// K2/std12k5/algoritms/YstavkiConfig
TYPE YstavkiConfig:
		{attribute 'symbol' := 'read'} 
	STRUCT
		blockkr1: (*REFERENCE TO*)  DiscretParametr (table:=ADR(YstTable)) ;//{name:блокировать самосдвиг крана 1}
		blockkr2:(*REFERENCE TO*) DiscretParametr (table:=ADR(YstTable));//{name:блокировать самосдвиг крана 2}
		blockkr3:(*REFERENCE TO*) DiscretParametr (table:=ADR(YstTable));//{name:блокировать самосдвиг крана 3}
		blockkr3b:(*REFERENCE TO*) DiscretParametr (table:=ADR(YstTable));//{name:блокировать самосдвиг крана 3б}
		blockkr4:(*REFERENCE TO*) DiscretParametr (table:=ADR(YstTable));//{name:блокировать самосдвиг крана 4}
		blockkr5:(*REFERENCE TO *)DiscretParametr (table:=ADR(YstTable));//{name:блокировать самосдвиг крана 5}
		blockkr6:(*REFERENCE TO *)DiscretParametr (table:=ADR(YstTable));//{name:блокировать самосдвиг крана 6}
		Block_kr4_alg:DiscretParametr (table:=ADR(YstTable));
		Block_kr1_alg:DiscretParametr (table:=ADR(YstTable));
		Block_kr2_alg:DiscretParametr (table:=ADR(YstTable));
		Block_kr3_alg:DiscretParametr (table:=ADR(YstTable));
		Block_kr3b_alg:DiscretParametr (table:=ADR(YstTable));
		Block_kr5_alg:DiscretParametr (table:=ADR(YstTable));
		Block_kr6_alg:DiscretParametr (table:=ADR(YstTable));
		
		block_OPC_cmd:DiscretParametr (table:=ADR(YstTable));
		
		////////////////////ПС по СИП//////////////////////////////////////////////////////
		SIp_T1: SIP_PS (table:=ADR(YstTable)):=(ai:= ai.TOpornogoPodshipnikaEDT_1);
		
		SIp_T2: SIP_PS (table:=ADR(YstTable)):=(ai:= ai.TOpornoYpornogoPodshipnikaEDT_2);
		
		SIp_T3: SIP_PS (table:=ADR(YstTable)):=(ai:= ai.TOpornoYpornogoPodshipnikaKolesaRedEDT_3);
		
		SIp_T4: SIP_PS (table:=ADR(YstTable)):=(ai:= ai.TOpornoYpornogoPodshipnikaKolesaRedHT_4);
		
		SIp_T5: SIP_PS (table:=ADR(YstTable)):=(ai:= ai.TOpornogoPodshipnikaShesterniReduktoraT_5);
		
		SIp_T6: SIP_PS (table:=ADR(YstTable)):=(ai:= ai.TOpornogoPodshipnikaReduktoraHT_6);
		
		SIp_T7_1: SIP_PS (table:=ADR(YstTable)):=(ai:= ai.TOpornoYpornogoPodshipnikaNagnetateljaT_7_1);
		
		SIp_T7_2: SIP_PS (table:=ADR(YstTable)):=(ai:= ai.TOpornoYpornogoPodshipnikaNagnetateljaT_7_2);
		
		SIp_T8_1: SIP_PS (table:=ADR(YstTable)):=(ai:= ai.TOpornoYpornogoPodshipnikaSvobodnogoKoncaNT_8_1);
		
		SIp_T8_2: SIP_PS (table:=ADR(YstTable)):=(ai:= ai.TOpornoYpornogoPodshipnikaSvobodnogoKoncaNT_8_2);
		
		SIp_T9_1: SIP_PS (table:=ADR(YstTable)):=(ai:= ai.TYpornogoPodshipnikaRavKolodokHT_9_1	);
		
		SIp_T9_2: SIP_PS (table:=ADR(YstTable)):=(ai:= ai.TYpornogoPodshipnikaRavKolodokHT_9_2	);
		
		SIp_T10_1: SIP_PS (table:=ADR(YstTable)):=(ai:= ai.TYpornogoPodshipnikaNerabKolodokHT_10_1	);
		
		SIp_T10_2: SIP_PS (table:=ADR(YstTable)):=(ai:= ai.TYpornogoPodshipnikaNerabKolodokHT_10_2	);
		
		SIp_T_Vyhode_N: SIP_PS (table:=ADR(YstTable)):=(ai:= ai.TgazaNaVyhodeH);
		
		SIp_T_Posle_AVOM: SIP_PS (table:=ADR(YstTable)):=(ai:= ai.TMaslaPosleAVOM);
		
		SIp_T_Masla_MB: SIP_PS (table:=ADR(YstTable)):=(ai:= ai.TMaslaMB);
		
		SIp_T_Masla_TEN: SIP_PS (table:=ADR(YstTable)):=(ai:= ai.TMaslaMB_TEN);
		
		////////////////////НАРАБОТКА//////////////////////////////////////////////////////
		
		nu1_narab: nu1 (table:=ADR(YstTable));		
		nu2_narab: nu2 (table:=ADR(YstTable));
		//pns_narab: pns_ (table:=ADR(YstTable));
		Work_HRS: work (table:=ADR(YstTable));
		Pusk_times: pusk (table:=ADR(YstTable));
		AO_times: AO (table:=ADR(YstTable));
		NO_times: NO (table:=ADR(YstTable));
		EO_times: EO (table:=ADR(YstTable));
		//CMN_Narab:CMN (table:=ADR(YstTable));
		//Kalorifer_AVOM_Narab: Kalorifer_AVOM (table:=ADR(YstTable));
		//TEN_Kollectora_narab: TEN_Kollectora (table:=ADR(YstTable));
	//	TEN_MB_Narab:			TEN_MB (table:=ADR(YstTable));
		////////////////////Уставки//////////////////////////////////////////////////////
		YstPNS_YP:  AutoPNS_YP (table:=ADR(YstTable));
		YstPNS_YT:  AutoPNS_YT (table:=ADR(YstTable));
		
		Yst_Vkl_TEN:	AutoTEN_YP (table:=ADR(YstTable));
		Yst_Vykl_TEN:	AutoTEN_YT (table:=ADR(YstTable));
		
		Yst_AVOM_T1:	T1_AVOM (table:=ADR(YstTable));
		Yst_AVOM_T2:	T2_AVOM (table:=ADR(YstTable));
		Yst_AVOM_T3:	T3_AVOM (table:=ADR(YstTable));
		Yst_AVOM_T4:	T4_AVOM (table:=ADR(YstTable));
		
		Yst_Tvkl_AVOM1:	Tvkl_AVOM1 (table:=ADR(YstTable));
		Yst_Tvkl_AVOM2:	Tvkl_AVOM2 (table:=ADR(YstTable));
		Yst_Tvkl_AVOM3:	Tvkl_AVOM3 (table:=ADR(YstTable));
		Yst_Tvkl_AVOM4:	Tvkl_AVOM4 (table:=ADR(YstTable));
		
		Yst_Tvykl_AVOM1:	Tvykl_AVOM1 (table:=ADR(YstTable));
		Yst_Tvykl_AVOM2:	Tvykl_AVOM2 (table:=ADR(YstTable));
		Yst_Tvykl_AVOM3:	Tvykl_AVOM3 (table:=ADR(YstTable));
		Yst_Tvykl_AVOM4:	Tvykl_AVOM4 (table:=ADR(YstTable));
		
		Yst_DTvykl_AVOM1:	Delta_Vykl_AVOM1 (table:=ADR(YstTable));
		Yst_DTvykl_AVOM2:	Delta_Vykl_AVOM2 (table:=ADR(YstTable));
		Yst_DTvykl_AVOM3:	Delta_Vykl_AVOM3 (table:=ADR(YstTable));
		Yst_DTvykl_AVOM4:	Delta_Vykl_AVOM4 (table:=ADR(YstTable));
		
		num_Avom:			Number_Of_Avom (table:=ADR(YstTable));
		
		////////////////////Управляющие сигналы//////////////////////////////////////////////////////
		//{name:рассогласование аналогов и дискрета по dPм-г}
		dPmg_Rassogl: Rassoglasovanie_dPmg (table:=ADR(YstTable)):=(di:=im.PerepadDavlenieMasloGaz_Less100, ai:=AI.PerepadDavlenieMasloGaz);
		dP_Konf_kr1:DiscretParametr (table:=ADR(YstTable));	
		dP_Konf_kr2:DiscretParametr (table:=ADR(YstTable));	
		(*sip_t1_new:SEt_New_SIP (table:=ADR(YstTable)):=(Ai:=ai.TOpornogoPodshipnikaEDT_1, n:= 0);*)
	END_STRUCT
END_TYPE

// lowLevel_ecl/kontroller/extSources/AnalogsProcessing
TYPE AnalogsProcessing :
(
	AVERAGEVALUE,
	MAXVALUE,
	MINVALUE,
	MEDIANVALUE
);
END_TYPE

// lowLevel_ecl/Common/table/TableDescriptor
TYPE TableDescriptor :
STRUCT
	head:POINTER TO BaseObject:=0;
	tail:POINTER TO BaseObject:=0;
END_STRUCT
END_TYPE

// lowLevel_ecl/im/sectionSwitch/basketStats
TYPE basketStats :
(
	BASKET_NOTDEFINED:=0,
	BASKET_ROLLEDIN:=1,
	BASKET_ROLLEDOUT:=2,
	BASKET_TRANSITIONAL:=3,
	BASKET_ERROR:=4,
	BASKET_TEST:=5
) BYTE;
END_TYPE

// lowLevel_ecl/kontroller/modbus/MbAiWordOrder
TYPE MbAiWordOrder :
(
	AiWordOrder12 := 0,
	AiWordOrder21 := 1
);
END_TYPE

// lowLevel_ecl/kontroller/modbus/MbKontrollerRole
TYPE MbKontrollerRole :
(
	MK_DONTKNOWN,
	MK_MASTER,
	MK_SLAVE
);
END_TYPE

// lowLevel_ecl/kontroller/modbus/Sources/FloatAsWords
TYPE FloatAsWords :
UNION
	fValue:REAL;
	wValue:ARRAY[0..1]OF WORD;
	dwValue:DWORD;
	bValue:ARRAY[0..4]OF BYTE;
END_UNION
END_TYPE

// lowLevel_ecl/kontroller/modbus/UsedByteMBSource
TYPE UsedByteMBSource :
(
	LB,
	HB
);
END_TYPE

// K1/std12k5/hardwareConfig/defines/hwC
	{attribute 'symbol' := 'readwrite'}
VAR_GLOBAL
	//SIP:	SIp_Yst (table:=0);
		{attribute 'symbol' := 'none'}
	kontrollers:TableDescriptor;
		{attribute 'symbol' := 'read'}
///	kontroller:elpk04(table:=ADR(kontrollers)):=(mlpConfig:='C:\\ELPK04\\Mlp2 2015-04-07\\MLP Projects\\1.mlp');
	kontroller:elpk04(table:=ADR(kontrollers)):=(mlpConfig:='\Storage Card\3s\RWHxxx.INI');// не должно находить такой файл никогда !!!
	di:DiConfig;
	ai:AiConfig;
	od:DOConfig;
	{attribute 'symbol' := 'none'}
	ao:AOConfig;
	//{attribute 'symbol' := 'none'}
	//mb:MbsConfig;

END_VAR

// K1/std12k5/logicConfig/defines/logicConfig
	{attribute 'symbol' := 'readwrite'}
VAR_GLOBAL
	{attribute 'symbol' := 'none'}
	imTable:TableDescriptor;
	
	{attribute 'symbol' := 'none'}
	iAmTrue:everifingTrue(table:=0);//Затычка из DiSource. Всегда возвращает одни и теже комбинации значения и достоверности
	OPC_Imit: Imit_OPC (table:=0);
	Im:ImConfig;
	{attribute 'symbol' := 'none'}
	Off_Q:All_Quation_Off (table:=0);
		{attribute 'symbol' := 'none'}
	PPU_Init_:PPU_Init (table:=0);
END_VAR

// K1/std12k5/algoritms/defines/algoritmsConf
	{attribute 'symbol' := 'readwrite'}
VAR_GLOBAL
	{attribute 'symbol' := 'none'}
	YstTable:TableDescriptor;
	Ystavki: YstavkiConfig;
	algManager:AlgoritmsManager(table:=0);
	algoritms:algoritmsConfig;
	{attribute 'symbol' := 'none'}
	protectManager:ProtectionManager (table:=0);
	protections:ProtectionsConfig;
	
	
END_VAR

// lowLevel_ecl/kontroller/mlp/FAUs
{attribute 'symbol' := 'none'}
VAR_GLOBAL
	
DIn_ 	:	ARRAY [0..255] 	OF DIn_s;		//	Сигнализация и неисправности дискретных входов (номер в массиве соответствует адресу конфигурации в MLP)
											//	f	:	WORD	;	//	bit-0 присутствие в проекте MLP. 1-есть, 0 -нет
																	//	bit-1 тип модуля 1-выходной, 0 -входной
																	//	bit-2 достоверность 1- достоверно,0- не достоверно 
											//	val	:	WORD	;	//	Контроль канала
																	//	Каждая цепь 2 бита
	                												//	00 - обыв цепи
																	//	01 - недостоверно
																	//	10 - контакт разомкнут
																	//	11 - контакт замкнут	

											//	DIn[63].val - меняющееся число для проверки связи с основным МЛП (задается в MLP)
											//	если	DIn[64].val = 7 - есть связь с BS-1 (задается в MLP)
											//	если	DIn[65].val = 7 - есть связь с BS-2 (задается в MLP)
											//	если	DIn[66].val = 7 - есть связь с BS-3 (задается в MLP)
											//	если	DIn[67].val = 7 - есть связь с BS-4 (задается в MLP)
																					
																	
AIn_ 	:	ARRAY [0..255] 	OF AIn_s;		//	Значение и неисправности аналоговых входов (номер в массиве соответствует адресу конфигурации в MLP)
											//	f	:	DWORD	;	//	bit-0 присутствие в проекте MLP. 1-есть, 0 –нет
																	//	bit-1 тип модуля 1-выходной, 0 -входной
																	//	bit-2 достоверность 1- достоверно,0- не достоверно. Диагностика общая: и по диапазонам измерения, и собственная по каналу модуля.
																	//	bit-3 размерность сигнала 1- в физических величинах,0- значение тока (0-20100)
																	//	bit-4 1- ниже нижней границы,0 - выше нижней границы
																	//	bit-5 1- выше верхней границы,0 - ниже верхней границы
																	//	bit-6 1- общий бит отказа канала( по ИЛИ Not(bit2), bit4, bit5)
											//	val	:	REAL	;	//	Значение аналогового входа 4-20мА - 40000-20000 

Dout_	:	ARRAY [0..255] 	OF WORD;		//	Массив дискретных выходов (один бит - один выход, одно слово - один модуль) (номер в массиве соответствует адресу конфигурации в MLP)
Din_Dout: 	ARRAY [0..255] 	OF sDIN_DOUT;	//	Массив неисправностей дискретных выходов
											//	s_Aux	:	WORD	;	//	bit-0 присутствие 1-есть, 0 -нет (привязка в конфигурации MLP)
																		//	bit-1 тип модуля 1-выходной, 0 -входной
																		//	bit-2 достоверность 1- достоверно,0- не достоверно
									  		//	kcc		:	WORD	;   //	Контроль Целостности Цепи - КЦЦ
																		//	каждая цепь 2 бита
																		//	00 - неизвестно или обрыв цепи
																		//	01 - есть Целостность Цепи
																		//	10 - есть ток
																		//	11 - КЗ
											//	kk		:	WORD	;	//	Контроль выхода команды - КК
																		//	каждая цепь 2 бита
																		//	00 - не бывает
																		//	01 - пассивное состояние
																		//	10 - активное (есть выход)состояние
																		//	11 - ошибка выхода команды 
									  		//	value_cc:	WORD	;	//	содержимое выходных регистров 

Aout_ 	:	ARRAY [0..255] 	OF REAL;		//	Массив аналоговых выходов (номер в массиве соответствует адресу конфигурации в MLP)
Ain_Aout:	ARRAY [0..255] 	OF sAIN_AOUT;	//	Массив неисправностей аналоговых выходов
											//	s_Aux	:	WORD	;	//	bit-0 присутствие 1-есть, 0 -нет
																		//	bit-1 тип модуля 1-выходной, 0 -входной
																		//	bit-2 достоверность 1- достоверно,0- не достоверно
																		//	s_value	:	REAL	;	//	Действительный (измеренный) выходной ток 4-20мА - 4000-20000

Diag_ 	:	ARRAY [0..63]	OF WORD;		//	массив неисправностей модулей
																		//	2 бита на 1 модуль
																		//	00 - ok
																		//	01 - нет модуля
																		//	10 - нулевые данные
																		//	11 - нет связи с модулем
END_VAR

// K1/std12k5/Elpk_03_02/GVL_COMMON
VAR_GLOBAL

//////////////////// П Е Р Е М Е Н Н Ы Е //////////////////////////////////////////////////////////////////////////////

	DI_K:ARRAY[0..255] OF T_DI03{WORD};
	AI_K:ARRAY[0..255] OF T_AI03{WORD};
	DO_K:ARRAY[0..255] OF T_DO03;
	
	MODULES03:ARRAY[1..16] OF T_DIAGNOSTIC03;
	IMIT_F:	WORD:= 0;	//16#55AA;







//	Глобальные переменные для резервирования
	H1:RTS_IEC_HANDLE;// pointer to byte
	S1:Com_Settings;
	S1ex:Com_SettingsEX;

	
//	Глобальные переменные для OPC
   {attribute 'displaymode':='hex'}
	BMPERR_I:WORD;		// внутреннее использование
   {attribute 'displaymode':='hex'}
	MxStatus_I:WORD;		// внутреннее использование
   {attribute 'displaymode':='hex'}
	MxMode_O:WORD;		// внутреннее использование
   {attribute 'displaymode':='hex'}
	BMPPRES_I:WORD;		// внутреннее использование






	



(*
//////////////////////////////////////////////////////////////////////
//This gobal variable list is received via the network.
//Sender: GVL2N_REZ [UP2: PLC Logic: Application]
//Protocol: UDP
//	Глобальные переменные для резервирования - это должно быть в глоб списке передачи К2
	PilaK2_O:WORD;
	StatusK2_O:WORD;
	ReadyK2_O:WORD;
////////////////////////////////////////////////////////////////////////
*)





//////////////////////////////////////////////////////////////////////
//This gobal variable list is received via the network.
//Sender: GVL1IMIT_to [Imitator1: PLC Logic: Application]
//Protocol: UDP
//	Глобальные переменные для моего имитатора. Должно быть в NVL1_from_IMIT
//
//
//   {attribute 'displaymode':='hex'}
//	Imitator_Code:WORD:=16#55AA;// код наличия имитатора - пересылается из имитатора в контроллеры!!!
   {attribute 'displaymode':='hex'}
	Imitator_Code:WORD:=16#0;// код наличия имитатора - пересылается из имитатора в контроллеры!!!

	// аналоговые входы нумеруем от 1
	AIs_Im:ARRAY[0..100] OF WORD;// рассылка из имитатора
	// дискретные входы нумеруем от 1
   {attribute 'displaymode':='hex'}
	DIs_Im:ARRAY[0..30] OF WORD;// рассылка из имитатора
(*
	// пока не используется в имитаторе !!!	
	// диагностика контроллера №1 
   {attribute 'displaymode':='hex'}
	NodeErr1_UP1_Im:WORD;// рассылка из имитатора
   {attribute 'displaymode':='hex'}
	NodeErr2_UP1_Im:WORD;// рассылка из имитатора
   {attribute 'displaymode':='hex'}
	NodeErr3_UP1_Im:WORD;// рассылка из имитатора
   {attribute 'displaymode':='hex'}
	NodeErr4_UP1_Im:WORD;// рассылка из имитатора
   {attribute 'displaymode':='hex'}
	NodeErr5_UP1_Im:WORD;// рассылка из имитатора
   {attribute 'displaymode':='hex'}
	NodeErr6_UP1_Im:WORD;// рассылка из имитатора
   {attribute 'displaymode':='hex'}
	NodeErr7_UP1_Im:WORD;// рассылка из имитатора
   {attribute 'displaymode':='hex'}
	NodeErr8_UP1_Im:WORD;// рассылка из имитатора
   {attribute 'displaymode':='hex'}
	NodeErr9_UP1_Im:WORD;// рассылка из имитатора
   {attribute 'displaymode':='hex'}
	NodeErr10_UP1_Im:WORD;// рассылка из имитатора
   {attribute 'displaymode':='hex'}
	NodeErr11_UP1_Im:WORD;// рассылка из имитатора
   {attribute 'displaymode':='hex'}
	NodeErr12_UP1_Im:WORD;// рассылка из имитатора
   {attribute 'displaymode':='hex'}
	NodeErr13_UP1_Im:WORD;// рассылка из имитатора
   {attribute 'displaymode':='hex'}
	NodeErr14_UP1_Im:WORD;// рассылка из имитатора
   {attribute 'displaymode':='hex'}
	NodeErr15_UP1_Im:WORD;// рассылка из имитатора
   {attribute 'displaymode':='hex'}
	NodeErr16_UP1_Im:WORD;// рассылка из имитатора
   {attribute 'displaymode':='hex'}
	BMPERR_UP1_Im:WORD;// рассылка из имитатора
   {attribute 'displaymode':='hex'}
	BMPPRES_UP1_Im:WORD;// рассылка из имитатора

	// диагностика контроллера №2 
   {attribute 'displaymode':='hex'}
	NodeErr1_UP2_Im:WORD;// рассылка из имитатора
   {attribute 'displaymode':='hex'}
	NodeErr2_UP2_Im:WORD;// рассылка из имитатора
   {attribute 'displaymode':='hex'}
	NodeErr3_UP2_Im:WORD;// рассылка из имитатора
   {attribute 'displaymode':='hex'}
	NodeErr4_UP2_Im:WORD;// рассылка из имитатора
   {attribute 'displaymode':='hex'}
	NodeErr5_UP2_Im:WORD;// рассылка из имитатора
   {attribute 'displaymode':='hex'}
	NodeErr6_UP2_Im:WORD;// рассылка из имитатора
   {attribute 'displaymode':='hex'}
	NodeErr7_UP2_Im:WORD;// рассылка из имитатора
   {attribute 'displaymode':='hex'}
	NodeErr8_UP2_Im:WORD;// рассылка из имитатора
   {attribute 'displaymode':='hex'}
	NodeErr9_UP2_Im:WORD;// рассылка из имитатора
   {attribute 'displaymode':='hex'}
	NodeErr10_UP2_Im:WORD;// рассылка из имитатора
   {attribute 'displaymode':='hex'}
	NodeErr11_UP2_Im:WORD;// рассылка из имитатора
   {attribute 'displaymode':='hex'}
	NodeErr12_UP2_Im:WORD;// рассылка из имитатора
   {attribute 'displaymode':='hex'}
	NodeErr13_UP2_Im:WORD;// рассылка из имитатора
   {attribute 'displaymode':='hex'}
	NodeErr14_UP2_Im:WORD;// рассылка из имитатора
   {attribute 'displaymode':='hex'}
	NodeErr15_UP2_Im:WORD;// рассылка из имитатора
   {attribute 'displaymode':='hex'}
	NodeErr16_UP2_Im:WORD;// рассылка из имитатора
   {attribute 'displaymode':='hex'}
	BMPERR_UP2_Im:WORD;// рассылка из имитатора
   {attribute 'displaymode':='hex'}
	BMPPRES_UP2_Im:WORD;// рассылка из имитатора
*)

END_VAR

// K1/std12k5/Elpk_03_02/GVL1N_REZ
VAR_GLOBAL
//	Глобальные переменные для резервирования
	PilaK1_O:WORD;
	StatusK1_O:WORD;
	ReadyK1_O:WORD;
		

END_VAR

// K1/std12k5/Elpk_03_02/GVLOPC
VAR_GLOBAL
//					
	LifeCnt:WORD;	// Пила жизни из контроллера: на каждом цикле +1 в диапазоне 0..1023
	
// диагностика контроллера	
   {attribute 'displaymode':='hex'}
	NodeErr1_K:WORD;	// OPC	
   {attribute 'displaymode':='hex'}
	NodeErr2_K:WORD;	// OPC
   {attribute 'displaymode':='hex'}
	NodeErr3_K:WORD;	// OPC
   {attribute 'displaymode':='hex'}
	NodeErr4_K:WORD;	// OPC
   {attribute 'displaymode':='hex'}
	NodeErr5_K:WORD;	// OPC
   {attribute 'displaymode':='hex'}
	NodeErr6_K:WORD;	// OPC
   {attribute 'displaymode':='hex'}
	NodeErr7_K:WORD;	// OPC
   {attribute 'displaymode':='hex'}
	NodeErr8_K:WORD;	// OPC
   {attribute 'displaymode':='hex'}
	NodeErr9_K:WORD;	// OPC
   {attribute 'displaymode':='hex'}
	NodeErr10_K:WORD;	// OPC
   {attribute 'displaymode':='hex'}
	NodeErr11_K:WORD;	// OPC
   {attribute 'displaymode':='hex'}
	NodeErr12_K:WORD;	// OPC
   {attribute 'displaymode':='hex'}
	NodeErr13_K:WORD;	// OPC
   {attribute 'displaymode':='hex'}
	NodeErr14_K:WORD;	// OPC
   {attribute 'displaymode':='hex'}
	NodeErr15_K:WORD;	// OPC
   {attribute 'displaymode':='hex'}
	NodeErr16_K:WORD;	// OPC

   {attribute 'displaymode':='hex'}
	CfgErr1_K:WORD;	// OPC	
   {attribute 'displaymode':='hex'}
	CfgErr2_K:WORD;	// OPC	
   {attribute 'displaymode':='hex'}
	CfgErr3_K:WORD;	// OPC	
   {attribute 'displaymode':='hex'}
	CfgErr4_K:WORD;	// OPC	
   {attribute 'displaymode':='hex'}
	CfgErr5_K:WORD;	// OPC	
   {attribute 'displaymode':='hex'}
	CfgErr6_K:WORD;	// OPC	
   {attribute 'displaymode':='hex'}
	CfgErr7_K:WORD;	// OPC	
   {attribute 'displaymode':='hex'}
	CfgErr8_K:WORD;	// OPC	
   {attribute 'displaymode':='hex'}
	CfgErr9_K:WORD;	// OPC	
   {attribute 'displaymode':='hex'}
	CfgErr10_K:WORD;	// OPC	
   {attribute 'displaymode':='hex'}
	CfgErr11_K:WORD;	// OPC	
   {attribute 'displaymode':='hex'}
	CfgErr12_K:WORD;	// OPC	
   {attribute 'displaymode':='hex'}
	CfgErr13_K:WORD;	// OPC	
   {attribute 'displaymode':='hex'}
	CfgErr14_K:WORD;	// OPC	
   {attribute 'displaymode':='hex'}
	CfgErr15_K:WORD;	// OPC	
   {attribute 'displaymode':='hex'}
	CfgErr16_K:WORD;	// OPC	




	
	
	
   {attribute 'displaymode':='hex'}
	BMPERR_K:WORD;	// OPC
   {attribute 'displaymode':='hex'}
	BMPPRES_K:WORD;	// OPC

   ///{attribute 'displaymode':='hex'}
	///DiagCnt_K:WORD;	// Пила диагностики из контроллера: на каждом цикле +1 в мл.байте и № контроллера в ст.байте
	
	
	
	// переменная master для ОРС-сервера
	MasterOPC_ST:BOOL;// ОРС-сервер читает переменную и если TRUE, то берет данные из этого контроллера
	LifeCntOPC:DWORD;// ОРС-сервер, если работает - записывает счетчик в переменную; если не работает- счетчик не изменяется




END_VAR

// K2/std12k5/hardwareConfig/defines/hwC
	{attribute 'symbol' := 'readwrite'}
VAR_GLOBAL
//	SIP:	SIp_Yst (table:=0);
		{attribute 'symbol' := 'none'}
	kontrollers:TableDescriptor;
		{attribute 'symbol' := 'read'}
///	kontroller:elpk04(table:=ADR(kontrollers)):=(mlpConfig:='C:\\ELPK04\\Mlp2 2015-04-07\\MLP Projects\\1.mlp');
	kontroller:elpk04(table:=ADR(kontrollers)):=(mlpConfig:='\Storage Card\3s\RWHxxx.INI');// не должно находить такой файл никогда !!!
	di:DiConfig;
	ai:AiConfig;
	od:DOConfig;
	{attribute 'symbol' := 'none'}
	ao:AOConfig;
//	{attribute 'symbol' := 'none'}
	//mb:MbsConfig;

END_VAR

// K2/std12k5/logicConfig/defines/logicConfig
	{attribute 'symbol' := 'readwrite'}
VAR_GLOBAL
	{attribute 'symbol' := 'none'}
	imTable:TableDescriptor;
	
	{attribute 'symbol' := 'none'}
	iAmTrue:everifingTrue(table:=0);//Затычка из DiSource. Всегда возвращает одни и теже комбинации значения и достоверности
	OPC_Imit: Imit_OPC (table:=0);
	Im:ImConfig;
	{attribute 'symbol' := 'none'}
	Off_Q:All_Quation_Off (table:=0);
		{attribute 'symbol' := 'none'}
	PPU_Init_:PPU_Init (table:=0);
END_VAR

// K2/std12k5/algoritms/defines/algoritmsConf
	{attribute 'symbol' := 'readwrite'}
VAR_GLOBAL
	{attribute 'symbol' := 'none'}
	YstTable:TableDescriptor;
	Ystavki: YstavkiConfig;
	algManager:AlgoritmsManager(table:=0);
	algoritms:algoritmsConfig;
	{attribute 'symbol' := 'none'}
	protectManager:ProtectionManager (table:=0);
	protections:ProtectionsConfig;
	
	
END_VAR

// K2/std12k5/Elpk_03_02/GVL_COMMON
VAR_GLOBAL

//////////////////// П Е Р Е М Е Н Н Ы Е //////////////////////////////////////////////////////////////////////////////

	DI_K:ARRAY[0..255] OF T_DI03{WORD};
	AI_K:ARRAY[0..255] OF T_AI03{WORD};
	DO_K:ARRAY[0..255] OF T_DO03;
	
	MODULES03:ARRAY[1..16] OF T_DIAGNOSTIC03;
	IMIT_F:	WORD:= 0;	//16#55AA;







//	Глобальные переменные для резервирования
	H1:RTS_IEC_HANDLE;// pointer to byte
	S1:Com_Settings;
	S1ex:Com_SettingsEX;

	
//	Глобальные переменные для OPC
   {attribute 'displaymode':='hex'}
	BMPERR_I:WORD;		// внутреннее использование
   {attribute 'displaymode':='hex'}
	MxStatus_I:WORD;		// внутреннее использование
   {attribute 'displaymode':='hex'}
	MxMode_O:WORD;		// внутреннее использование
   {attribute 'displaymode':='hex'}
	BMPPRES_I:WORD;		// внутреннее использование






	



(*
//////////////////////////////////////////////////////////////////////
//This gobal variable list is received via the network.
//Sender: GVL2N_REZ [UP2: PLC Logic: Application]
//Protocol: UDP
//	Глобальные переменные для резервирования - это должно быть в глоб списке передачи К2
	PilaK2_O:WORD;
	StatusK2_O:WORD;
	ReadyK2_O:WORD;
////////////////////////////////////////////////////////////////////////
*)





//////////////////////////////////////////////////////////////////////
//This gobal variable list is received via the network.
//Sender: GVL1IMIT_to [Imitator1: PLC Logic: Application]
//Protocol: UDP
//	Глобальные переменные для моего имитатора. Должно быть в NVL1_from_IMIT
//
//
//   {attribute 'displaymode':='hex'}
//	Imitator_Code:WORD:=16#55AA;// код наличия имитатора - пересылается из имитатора в контроллеры!!!
   {attribute 'displaymode':='hex'}
	Imitator_Code:WORD:=16#0;// код наличия имитатора - пересылается из имитатора в контроллеры!!!

	// аналоговые входы нумеруем от 1
	AIs_Im:ARRAY[0..100] OF WORD;// рассылка из имитатора
	// дискретные входы нумеруем от 1
   {attribute 'displaymode':='hex'}
	DIs_Im:ARRAY[0..30] OF WORD;// рассылка из имитатора
(*
	// пока не используется в имитаторе !!!	
	// диагностика контроллера №1 
   {attribute 'displaymode':='hex'}
	NodeErr1_UP1_Im:WORD;// рассылка из имитатора
   {attribute 'displaymode':='hex'}
	NodeErr2_UP1_Im:WORD;// рассылка из имитатора
   {attribute 'displaymode':='hex'}
	NodeErr3_UP1_Im:WORD;// рассылка из имитатора
   {attribute 'displaymode':='hex'}
	NodeErr4_UP1_Im:WORD;// рассылка из имитатора
   {attribute 'displaymode':='hex'}
	NodeErr5_UP1_Im:WORD;// рассылка из имитатора
   {attribute 'displaymode':='hex'}
	NodeErr6_UP1_Im:WORD;// рассылка из имитатора
   {attribute 'displaymode':='hex'}
	NodeErr7_UP1_Im:WORD;// рассылка из имитатора
   {attribute 'displaymode':='hex'}
	NodeErr8_UP1_Im:WORD;// рассылка из имитатора
   {attribute 'displaymode':='hex'}
	NodeErr9_UP1_Im:WORD;// рассылка из имитатора
   {attribute 'displaymode':='hex'}
	NodeErr10_UP1_Im:WORD;// рассылка из имитатора
   {attribute 'displaymode':='hex'}
	NodeErr11_UP1_Im:WORD;// рассылка из имитатора
   {attribute 'displaymode':='hex'}
	NodeErr12_UP1_Im:WORD;// рассылка из имитатора
   {attribute 'displaymode':='hex'}
	NodeErr13_UP1_Im:WORD;// рассылка из имитатора
   {attribute 'displaymode':='hex'}
	NodeErr14_UP1_Im:WORD;// рассылка из имитатора
   {attribute 'displaymode':='hex'}
	NodeErr15_UP1_Im:WORD;// рассылка из имитатора
   {attribute 'displaymode':='hex'}
	NodeErr16_UP1_Im:WORD;// рассылка из имитатора
   {attribute 'displaymode':='hex'}
	BMPERR_UP1_Im:WORD;// рассылка из имитатора
   {attribute 'displaymode':='hex'}
	BMPPRES_UP1_Im:WORD;// рассылка из имитатора

	// диагностика контроллера №2 
   {attribute 'displaymode':='hex'}
	NodeErr1_UP2_Im:WORD;// рассылка из имитатора
   {attribute 'displaymode':='hex'}
	NodeErr2_UP2_Im:WORD;// рассылка из имитатора
   {attribute 'displaymode':='hex'}
	NodeErr3_UP2_Im:WORD;// рассылка из имитатора
   {attribute 'displaymode':='hex'}
	NodeErr4_UP2_Im:WORD;// рассылка из имитатора
   {attribute 'displaymode':='hex'}
	NodeErr5_UP2_Im:WORD;// рассылка из имитатора
   {attribute 'displaymode':='hex'}
	NodeErr6_UP2_Im:WORD;// рассылка из имитатора
   {attribute 'displaymode':='hex'}
	NodeErr7_UP2_Im:WORD;// рассылка из имитатора
   {attribute 'displaymode':='hex'}
	NodeErr8_UP2_Im:WORD;// рассылка из имитатора
   {attribute 'displaymode':='hex'}
	NodeErr9_UP2_Im:WORD;// рассылка из имитатора
   {attribute 'displaymode':='hex'}
	NodeErr10_UP2_Im:WORD;// рассылка из имитатора
   {attribute 'displaymode':='hex'}
	NodeErr11_UP2_Im:WORD;// рассылка из имитатора
   {attribute 'displaymode':='hex'}
	NodeErr12_UP2_Im:WORD;// рассылка из имитатора
   {attribute 'displaymode':='hex'}
	NodeErr13_UP2_Im:WORD;// рассылка из имитатора
   {attribute 'displaymode':='hex'}
	NodeErr14_UP2_Im:WORD;// рассылка из имитатора
   {attribute 'displaymode':='hex'}
	NodeErr15_UP2_Im:WORD;// рассылка из имитатора
   {attribute 'displaymode':='hex'}
	NodeErr16_UP2_Im:WORD;// рассылка из имитатора
   {attribute 'displaymode':='hex'}
	BMPERR_UP2_Im:WORD;// рассылка из имитатора
   {attribute 'displaymode':='hex'}
	BMPPRES_UP2_Im:WORD;// рассылка из имитатора
*)

END_VAR

// K2/std12k5/Elpk_03_02/GVL2N_REZ
VAR_GLOBAL
//	Глобальные переменные для резервирования
	PilaK2_O:WORD;
	StatusK2_O:WORD;
	ReadyK2_O:WORD;
		

END_VAR

// K2/std12k5/Elpk_03_02/GVLOPC
VAR_GLOBAL
//					
	LifeCnt:WORD;	// Пила жизни из контроллера: на каждом цикле +1 в диапазоне 0..1023
	
// диагностика контроллера	
   {attribute 'displaymode':='hex'}
	NodeErr1_K:WORD;	// OPC	
   {attribute 'displaymode':='hex'}
	NodeErr2_K:WORD;	// OPC
   {attribute 'displaymode':='hex'}
	NodeErr3_K:WORD;	// OPC
   {attribute 'displaymode':='hex'}
	NodeErr4_K:WORD;	// OPC
   {attribute 'displaymode':='hex'}
	NodeErr5_K:WORD;	// OPC
   {attribute 'displaymode':='hex'}
	NodeErr6_K:WORD;	// OPC
   {attribute 'displaymode':='hex'}
	NodeErr7_K:WORD;	// OPC
   {attribute 'displaymode':='hex'}
	NodeErr8_K:WORD;	// OPC
   {attribute 'displaymode':='hex'}
	NodeErr9_K:WORD;	// OPC
   {attribute 'displaymode':='hex'}
	NodeErr10_K:WORD;	// OPC
   {attribute 'displaymode':='hex'}
	NodeErr11_K:WORD;	// OPC
   {attribute 'displaymode':='hex'}
	NodeErr12_K:WORD;	// OPC
   {attribute 'displaymode':='hex'}
	NodeErr13_K:WORD;	// OPC
   {attribute 'displaymode':='hex'}
	NodeErr14_K:WORD;	// OPC
   {attribute 'displaymode':='hex'}
	NodeErr15_K:WORD;	// OPC
   {attribute 'displaymode':='hex'}
	NodeErr16_K:WORD;	// OPC

   {attribute 'displaymode':='hex'}
	CfgErr1_K:WORD;	// OPC	
   {attribute 'displaymode':='hex'}
	CfgErr2_K:WORD;	// OPC	
   {attribute 'displaymode':='hex'}
	CfgErr3_K:WORD;	// OPC	
   {attribute 'displaymode':='hex'}
	CfgErr4_K:WORD;	// OPC	
   {attribute 'displaymode':='hex'}
	CfgErr5_K:WORD;	// OPC	
   {attribute 'displaymode':='hex'}
	CfgErr6_K:WORD;	// OPC	
   {attribute 'displaymode':='hex'}
	CfgErr7_K:WORD;	// OPC	
   {attribute 'displaymode':='hex'}
	CfgErr8_K:WORD;	// OPC	
   {attribute 'displaymode':='hex'}
	CfgErr9_K:WORD;	// OPC	
   {attribute 'displaymode':='hex'}
	CfgErr10_K:WORD;	// OPC	
   {attribute 'displaymode':='hex'}
	CfgErr11_K:WORD;	// OPC	
   {attribute 'displaymode':='hex'}
	CfgErr12_K:WORD;	// OPC	
   {attribute 'displaymode':='hex'}
	CfgErr13_K:WORD;	// OPC	
   {attribute 'displaymode':='hex'}
	CfgErr14_K:WORD;	// OPC	
   {attribute 'displaymode':='hex'}
	CfgErr15_K:WORD;	// OPC	
   {attribute 'displaymode':='hex'}
	CfgErr16_K:WORD;	// OPC	




	
	
	
   {attribute 'displaymode':='hex'}
	BMPERR_K:WORD;	// OPC
   {attribute 'displaymode':='hex'}
	BMPPRES_K:WORD;	// OPC

   ///{attribute 'displaymode':='hex'}
	///DiagCnt_K:WORD;	// Пила диагностики из контроллера: на каждом цикле +1 в мл.байте и № контроллера в ст.байте
	
	
	
	// переменная master для ОРС-сервера
	MasterOPC_ST:BOOL;// ОРС-сервер читает переменную и если TRUE, то берет данные из этого контроллера
	LifeCntOPC:DWORD;// ОРС-сервер, если работает - записывает счетчик в переменную; если не работает- счетчик не изменяется




END_VAR

// K1/std12k5/Elpk_03_02/NVL1_REZ
//This gobal variable list is received via the network.
//Sender: GVL2N_REZ [K2: PLC Logic: std12k5]
//Protocol: UDP

VAR_GLOBAL
//	Глобальные переменные для резервирования
	PilaK2_O:WORD;
	StatusK2_O:WORD;
	ReadyK2_O:WORD;
		

END_VAR

// K2/std12k5/Elpk_03_02/NVL2_REZ
//This gobal variable list is received via the network.
//Sender: GVL1N_REZ [K1: PLC Logic: std12k5]
//Protocol: UDP

VAR_GLOBAL
//	Глобальные переменные для резервирования
	PilaK1_O:WORD;
	StatusK1_O:WORD;
	ReadyK1_O:WORD;
		

END_VAR

// K1/std12k5/MAIN
PROGRAM MAIN
VAR

END_VAR


ELPK03_to_MLP_IN();// читать входы ЭЛПК-03-02 и передать в массивы 04

MainUP_PRG();// диагностика и OPC


///////////////////////////////////////////////////////////////////////////////////////////////////////////////////////
callExec(kontrollers);

{IF defined(imit)}
	{warning 'РЕЖИМ ИМИТАЦИИ! Входы и выходы отключены от физического источника'}
{ELSE}
execKontrollersInputs(table:=kontrollers);
{END_IF}

//SIP ();
callExec (YstTable);
callExec(imTable);
ProtectManager ();
OPC_Imit ();
algManager();
PPU_Init_ ();
Off_Q ();
{IF NOT defined(imit)}
execKontrollersOutputs(table:=kontrollers);
{END_IF}
///////////////////////////////////////////////////////////////////////////////////////////////////////////////////////

ELPK03_to_MLP_OUT(DO2_BLK:= 16#FF00, DO3_BLK:= 16#18FF);	// читать массивы 04 и передать в выходы ЭЛПК-03-02
										// с блокировкой ст байта DO_K[2] для индикации резервирования
										// с блокировкой мл байта DO_K[3] (сигналы резервирования старого) + DO_K[3].11 + DO_K[3].12 (индикация активности К1 и К2)

END_PROGRAM

// Elpk_03_02_COMMON/ELPK03_to_MLP_IN
PROGRAM ELPK03_to_MLP_IN
VAR
	I:INT;
END_VAR

	// переменные ы формате MLP			// переменные в формате ЭЛПК-03-02

	FOR I:=0 TO 24 DO
		///DI_K[I].Im := DIs_Im[I];// [0..30]
		IF (Imitator_Code=16#55AA)
		THEN// имитатор вкл
			DI_K[I].Imx := Imitator_Code{IMIT_F};
			DI_K[I].RR := DI_K[I].Im;
			DI_K[I].VeraB:= TRUE; 
		ELSE
			DI_K[I].Imx := 0;
			DI_K[I].RR := DI_K[I].In;
		END_IF
	END_FOR
	FOR I:=0 TO 71 DO
		///AI_K[I].Im := AIs_Im[I];// [0..100]
		IF (Imitator_Code=16#55AA)
		THEN// имитатор вкл
			AI_K[I].Imx := Imitator_Code{IMIT_F};
			AI_K[I].RR := AI_K[I].Im;
			AI_K[I].VeraB:= TRUE;
		ELSE
			AI_K[I].Imx := 0;
			AI_K[I].RR := AI_K[I].In;
		END_IF
	END_FOR

	//	MXIN	поз.1
	DI_K[0].VeraB:=		DI_K[0].Vera.0; 
	DI_K[1].VeraB:=		DI_K[0].Vera.1; 
	DI_K[2].VeraB:=		DI_K[0].Vera.2; 
	DI_K[3].VeraB:=		DI_K[0].Vera.3; 
	DI_K[4].VeraB:=		DI_K[0].Vera.4; 
	DI_K[5].VeraB:=		DI_K[0].Vera.5; 
	DI_K[6].VeraB:=		DI_K[0].Vera.6; 
	DI_K[7].VeraB:=		DI_K[0].Vera.7; 
	DI_K[8].VeraB:=		DI_K[0].Vera.8; 
	DI_K[9].VeraB:=		DI_K[0].Vera.9; 
	DI_K[10].VeraB:=	DI_K[0].Vera.10; 
	DI_K[11].VeraB:=	DI_K[0].Vera.11; 
	DI_K[12].VeraB:=	DI_K[0].Vera.12; 
	DI_K[13].VeraB:=	DI_K[0].Vera.13; 
	//	DIN	поз.8
	DI_K[14].VeraB:=	DI_K[14].Vera <> 0; 
	//	DIN	поз.10
	DI_K[15].VeraB:=	DI_K[15].Vera <> 0; 
	
	

	//	AIN	поз.15
	AI_K[0].VeraB:=		AI_K[0].Vera.0;
	AI_K[1].VeraB:=		AI_K[0].Vera.1;
	AI_K[2].VeraB:=		AI_K[0].Vera.2;
	AI_K[3].VeraB:=		AI_K[0].Vera.3;
	AI_K[4].VeraB:=		AI_K[0].Vera.4;
	AI_K[5].VeraB:=		AI_K[0].Vera.5;
	AI_K[6].VeraB:=		AI_K[0].Vera.6;
	AI_K[7].VeraB:=		AI_K[0].Vera.7;
	AI_K[8].VeraB:=		AI_K[0].Vera.8;
	AI_K[9].VeraB:=		AI_K[0].Vera.9;
	AI_K[10].VeraB:=	AI_K[0].Vera.10;
	AI_K[11].VeraB:=	AI_K[0].Vera.11;
	AI_K[12].VeraB:=	AI_K[0].Vera.12;
	AI_K[13].VeraB:=	AI_K[0].Vera.13;
	AI_K[14].VeraB:=	AI_K[0].Vera.14;
	AI_K[15].VeraB:=	AI_K[0].Vera.15;
	//	AIN	поз.13
	AI_K[16].VeraB:=	AI_K[16].Vera.0; 
	AI_K[17].VeraB:=	AI_K[16].Vera.1; 
	AI_K[18].VeraB:=	AI_K[16].Vera.2; 
	AI_K[19].VeraB:=	AI_K[16].Vera.3; 
	AI_K[20].VeraB:=	AI_K[16].Vera.4; 
	AI_K[21].VeraB:=	AI_K[16].Vera.5; 
	AI_K[22].VeraB:=	AI_K[16].Vera.6; 
	AI_K[23].VeraB:=	AI_K[16].Vera.7; 
	AI_K[24].VeraB:=	AI_K[16].Vera.8; 
	AI_K[25].VeraB:=	AI_K[16].Vera.9; 
	AI_K[26].VeraB:=	AI_K[16].Vera.10; 
	AI_K[27].VeraB:=	AI_K[16].Vera.11; 
	AI_K[28].VeraB:=	AI_K[16].Vera.12; 
	AI_K[29].VeraB:=	AI_K[16].Vera.13; 
	AI_K[30].VeraB:=	AI_K[16].Vera.14; 
	AI_K[31].VeraB:=	AI_K[16].Vera.15; 
	//	AIN	поз.11
	AI_K[32].VeraB:=	AI_K[32].Vera.0; 
	AI_K[33].VeraB:=	AI_K[32].Vera.1; 
	AI_K[34].VeraB:=	AI_K[32].Vera.2; 
	AI_K[35].VeraB:=	AI_K[32].Vera.3; 
	AI_K[36].VeraB:=	AI_K[32].Vera.4; 
	AI_K[37].VeraB:=	AI_K[32].Vera.5; 
	AI_K[38].VeraB:=	AI_K[32].Vera.6; 
	AI_K[39].VeraB:=	AI_K[32].Vera.7; 
	//	AIN	поз.9
	AI_K[40].VeraB:=	AI_K[40].Vera.0; 
	AI_K[41].VeraB:=	AI_K[40].Vera.1; 
	AI_K[42].VeraB:=	AI_K[40].Vera.2; 
	AI_K[43].VeraB:=	AI_K[40].Vera.3; 
	AI_K[44].VeraB:=	AI_K[40].Vera.4; 
	AI_K[45].VeraB:=	AI_K[40].Vera.5; 
	AI_K[46].VeraB:=	AI_K[40].Vera.6; 
	AI_K[47].VeraB:=	AI_K[40].Vera.7; 
	//	AIN	поз.16
	AI_K[48].VeraB:=	AI_K[48].Vera.0; 
	AI_K[49].VeraB:=	AI_K[48].Vera.1; 
	AI_K[50].VeraB:=	AI_K[48].Vera.2; 
	AI_K[51].VeraB:=	AI_K[48].Vera.3; 
	AI_K[52].VeraB:=	AI_K[48].Vera.4; 
	AI_K[53].VeraB:=	AI_K[48].Vera.5; 
	AI_K[54].VeraB:=	AI_K[48].Vera.6; 
	AI_K[55].VeraB:=	AI_K[48].Vera.7; 
	//	AIN	поз.14
	AI_K[56].VeraB:=	AI_K[56].Vera.0; 
	AI_K[57].VeraB:=	AI_K[56].Vera.1; 
	AI_K[58].VeraB:=	AI_K[56].Vera.2; 
	AI_K[59].VeraB:=	AI_K[56].Vera.3; 
	AI_K[60].VeraB:=	AI_K[56].Vera.4; 
	AI_K[61].VeraB:=	AI_K[56].Vera.5; 
	AI_K[62].VeraB:=	AI_K[56].Vera.6; 
	AI_K[63].VeraB:=	AI_K[56].Vera.7; 
	//	AIN	поз.12
	AI_K[64].VeraB:=	AI_K[64].Vera.0; 
	AI_K[65].VeraB:=	AI_K[64].Vera.1; 
	AI_K[66].VeraB:=	AI_K[64].Vera.2; 
	AI_K[67].VeraB:=	AI_K[64].Vera.3; 
	AI_K[68].VeraB:=	AI_K[64].Vera.4; 
	AI_K[69].VeraB:=	AI_K[64].Vera.5; 
	AI_K[70].VeraB:=	AI_K[64].Vera.6; 
	AI_K[71].VeraB:=	AI_K[64].Vera.7; 

	
	
	//******************************************************************************************************************************
	//	ЭЛПК-04		:	дискретный ввод через T12S44
	//******************************************************************************************************************************
	kontroller.DIn_[0].f		:= 5;	// .0 - есть в проекте		.1 - входные		.2 - достоверность		
	kontroller.DIn_[0].f.2		:= DI_K[0].VeraB;	// достоверность из драйвера RWH (=1 - достоверно)	
	//kontroller.DIn_[0].f.2		:= (kontroller.DIn_[0].val.1=0);		// недостоверность - получим их NodeErr модуля ???		
	//
	//	сигнал: Кран 1 открыт					обрыв: Нет обрыва
	DI_03_R	(N_Pair:=1, DI_K0:= DI_K[0].RR.0,	DIb_K0:= 1,					K_OUT:= kontroller.DIn_[0].val);
	//	сигнал: Кран 1 закрыт					обрыв: Нет обрыва
	DI_03_R	(N_Pair:=2, DI_K0:= DI_K[0].RR.1,	DIb_K0:= 1,					K_OUT:= kontroller.DIn_[0].val);
	// сигнал: Кран 2 открыт					обрыв: Нет обрыва
	DI_03_R	(N_Pair:=3, DI_K0:= DI_K[0].RR.2,	DIb_K0:= 1,					K_OUT:= kontroller.DIn_[0].val);
	//	сигнал: Кран 2 закрыт					обрыв: Нет обрыва
	DI_03_R	(N_Pair:=4, DI_K0:= DI_K[0].RR.3,	DIb_K0:= 1,					K_OUT:= kontroller.DIn_[0].val);
	//	сигнал: Кран 3 открыт					обрыв: Нет обрыва
	DI_03_R	(N_Pair:=5, DI_K0:= DI_K[0].RR.4,	DIb_K0:= 1,					K_OUT:= kontroller.DIn_[0].val);
	//	сигнал: Кран 3 закрыт					обрыв: Нет обрыва
	DI_03_R	(N_Pair:=6, DI_K0:= DI_K[0].RR.5,	DIb_K0:= 1,					K_OUT:= kontroller.DIn_[0].val);
	//	сигнал: Кран 3бис открыт				обрыв: Нет обрыва
	DI_03_R	(N_Pair:=7, DI_K0:= DI_K[0].RR.6,	DIb_K0:= 1,					K_OUT:= kontroller.DIn_[0].val);
	//	сигнал: Кран 3бис закрыт				обрыв: Нет обрыва
	DI_03_R	(N_Pair:=8, DI_K0:= DI_K[0].RR.7,	DIb_K0:= 1,					K_OUT:= kontroller.DIn_[0].val);
	
	
	kontroller.DIn_[1].f		:= 5;	// .0 - есть в проекте		.1 - входные		.2 - достоверность		
	kontroller.DIn_[1].f.2		:= DI_K[0].VeraB;	// достоверность из драйвера RWH (=1 - достоверно)	
	//kontroller.DIn_[1].f.2		:= (kontroller.DIn_[0].val.1=0);		// недостоверность - получим их NodeErr модуля ???		
	//
	//	сигнал: Кран 4 открыт					обрыв: Нет обрыва
	DI_03_R	(N_Pair:=1, DI_K0:= DI_K[0].RR.8,	DIb_K0:= 1,					K_OUT:= kontroller.DIn_[1].val);
	//	сигнал: Кран 4 закрыт					обрыв: Нет обрыва
	DI_03_R	(N_Pair:=2, DI_K0:= DI_K[0].RR.9,	DIb_K0:= 1,					K_OUT:= kontroller.DIn_[1].val);
	//	сигнал: Кран 5 открыт					обрыв: Нет обрыва
	DI_03_R	(N_Pair:=3, DI_K0:= DI_K[0].RR.10,	DIb_K0:= 1,					K_OUT:= kontroller.DIn_[1].val);
	//	сигнал: Кран 5 закрыт					обрыв: Нет обрыва
	DI_03_R	(N_Pair:=4, DI_K0:= DI_K[0].RR.11,	DIb_K0:= 1,					K_OUT:= kontroller.DIn_[1].val);
	//	сигнал: Кран 6 открыт					обрыв: Нет обрыва
	DI_03_R	(N_Pair:=5, DI_K0:= DI_K[0].RR.12,	DIb_K0:= 1,					K_OUT:= kontroller.DIn_[1].val);
	//	сигнал: Кран 6 закрыт					обрыв: Нет обрыва
	DI_03_R	(N_Pair:=6, DI_K0:= DI_K[0].RR.13,	DIb_K0:= 1,					K_OUT:= kontroller.DIn_[1].val);
	// сигнал: Не подключено					обрыв: Не подключено
	DI_03_R	(N_Pair:=7, DI_K0:= 0,				DIb_K0:= 0,					K_OUT:= kontroller.DIn_[1].val);
	// сигнал: Не подключено					обрыв: Не подключено
	DI_03_R	(N_Pair:=8, DI_K0:= 0,				DIb_K0:= 0,					K_OUT:= kontroller.DIn_[1].val);
	
	
	kontroller.DIn_[2].f		:= 5;	// .0 - есть в проекте		.1 - входные		.2 - достоверность		
	kontroller.DIn_[2].f.2		:= DI_K[1].VeraB;	// достоверность из драйвера RWH (=1 - достоверно)	
	//kontroller.DIn_[2].f.2		:= (kontroller.DIn_[0].val.1=0);		// недостоверность - получим их NodeErr модуля ???		
	//
	// сигнал: АВО масла №1 в авт. режиме		обрыв: Нет обрыва
	DI_03_R	(N_Pair:=1, DI_K0:= DI_K[1].RR.0,	DIb_K0:= 1,					K_OUT:= kontroller.DIn_[2].val);
	// сигнал: АВО масла №2 в авт. режиме		обрыв: Нет обрыва
	DI_03_R	(N_Pair:=2, DI_K0:= DI_K[1].RR.1,	DIb_K0:= 1,					K_OUT:= kontroller.DIn_[2].val);
	// сигнал: АВО масла №3 в авт. режиме		обрыв: Нет обрыва
	DI_03_R	(N_Pair:=3, DI_K0:= DI_K[1].RR.2,	DIb_K0:= 1,					K_OUT:= kontroller.DIn_[2].val);
	// сигнал: АВО масла №4 в авт. режиме		обрыв: Нет обрыва
	DI_03_R	(N_Pair:=4, DI_K0:= DI_K[1].RR.3,	DIb_K0:= 1,					K_OUT:= kontroller.DIn_[2].val);
	// сигнал: ПНС в автоматическом режиме		обрыв: Нет обрыва
	DI_03_R	(N_Pair:=5, DI_K0:= DI_K[1].RR.4,	DIb_K0:= 1,					K_OUT:= kontroller.DIn_[2].val);
	// сигнал: НУ1 в автоматическом режиме		обрыв: Нет обрыва
	DI_03_R	(N_Pair:=6, DI_K0:= DI_K[1].RR.5,	DIb_K0:= 1,					K_OUT:= kontroller.DIn_[2].val);
	// сигнал: НУ2 в автоматическом режиме		обрыв: Нет обрыва
	DI_03_R	(N_Pair:=7, DI_K0:= DI_K[1].RR.6,	DIb_K0:= 1,					K_OUT:= kontroller.DIn_[2].val);
	// сигнал: ТЭН маслобака в авт. режиме		обрыв: Нет обрыва
	DI_03_R	(N_Pair:=8, DI_K0:= DI_K[1].RR.7,	DIb_K0:= 1,					K_OUT:= kontroller.DIn_[2].val);

	
	kontroller.DIn_[3].f		:= 5;	// .0 - есть в проекте		.1 - входные		.2 - достоверность		
	kontroller.DIn_[3].f.2		:= DI_K[1].VeraB;	// достоверность из драйвера RWH (=1 - достоверно)	
	//kontroller.DIn_[3].f.2		:= (kontroller.DIn_[0].val.1=0);		// недостоверность - получим их NodeErr модуля ???		
	//
	// сигнал: Подогреватель коллектора в авт. режиме		обрыв: Нет обрыва
	DI_03_R	(N_Pair:=1, DI_K0:= DI_K[1].RR.8,				DIb_K0:= 1,					K_OUT:= kontroller.DIn_[3].val);
	// сигнал: Калорифер АВО масла в авт. режиме			обрыв: Нет обрыва
	DI_03_R	(N_Pair:=2, DI_K0:= DI_K[1].RR.9,				DIb_K0:= 1,					K_OUT:= kontroller.DIn_[3].val);
	// сигнал: Циркуляционный насос в авт. режиме			обрыв: Нет обрыва
	DI_03_R	(N_Pair:=3, DI_K0:= DI_K[1].RR.10,				DIb_K0:= 1,					K_OUT:= kontroller.DIn_[3].val);
	// сигнал: Не подключено								обрыв: Не подключено
	DI_03_R	(N_Pair:=4, DI_K0:= DI_K[1].RR.11,				DIb_K0:= 1,					K_OUT:= kontroller.DIn_[3].val);
	// сигнал: Синхронизация режима К2						обрыв: Нет обрыва
	DI_03_R	(N_Pair:=5, DI_K0:= DI_K[1].RR.12,				DIb_K0:= 1,					K_OUT:= kontroller.DIn_[3].val);
	// сигнал: Синхронизация режима К1						обрыв: Нет обрыва
	DI_03_R	(N_Pair:=6, DI_K0:= DI_K[1].RR.13,				DIb_K0:= 1,					K_OUT:= kontroller.DIn_[3].val);
	// сигнал: Не подключено								обрыв: Не подключено
	DI_03_R	(N_Pair:=7, DI_K0:= 0,							DIb_K0:= 0,					K_OUT:= kontroller.DIn_[3].val);
	// сигнал: Не подключено								обрыв: Не подключено
	DI_03_R	(N_Pair:=8, DI_K0:= 0,							DIb_K0:= 0,					K_OUT:= kontroller.DIn_[3].val);
	

	kontroller.DIn_[4].f		:= 5;	// .0 - есть в проекте		.1 - входные		.2 - достоверность		
	kontroller.DIn_[4].f.2		:= DI_K[2].VeraB;	// достоверность из драйвера RWH (=1 - достоверно)	
	//kontroller.DIn_[4].f.2		:= (kontroller.DIn_[0].val.1=0);		// недостоверность - получим их NodeErr модуля ???		
	//
	// сигнал: dP масло-газ < 100 кПА			обрыв:  dP масло-газ < 100 кПА
	DI_03_R	(N_Pair:=1, DI_K0:= DI_K[2].RR.0,	DIb_K0:= DI_K[2].RR.1,			K_OUT:= kontroller.DIn_[4].val);
	// сигнал: dP газа на КР1 > 100 кПА			обрыв:  dP газа на КР1 > 100 кПА
	DI_03_R	(N_Pair:=2, DI_K0:= DI_K[2].RR.2,	DIb_K0:= DI_K[2].RR.3,			K_OUT:= kontroller.DIn_[4].val);
	// сигнал: Отклонение уровня масла в АКК уплотнения		обрыв:  Отклонение уровня масла в АКК уплотнения
	DI_03_R	(N_Pair:=3, DI_K0:= DI_K[2].RR.4,	DIb_K0:= DI_K[2].RR.5,			K_OUT:= kontroller.DIn_[4].val);
	// сигнал: Загазованность двигателя 0.5% (РЕЗЕРВ)		обрыв:  Загазованность двигателя 0.5% (РЕЗЕРВ)
	DI_03_R	(N_Pair:=4, DI_K0:= DI_K[2].RR.6,	DIb_K0:= DI_K[2].RR.7,			K_OUT:= kontroller.DIn_[4].val);
	// сигнал: Загазованность двигателя 1.0% (РЕЗЕРВ)		обрыв:  Загазованность двигателя 1.0% (РЕЗЕРВ)
	DI_03_R	(N_Pair:=5, DI_K0:= DI_K[2].RR.8,	DIb_K0:= DI_K[2].RR.9,			K_OUT:= kontroller.DIn_[4].val);
	// сигнал: Загазованность нагнетателя 0.5% (РЕЗЕРВ)		обрыв:  Загазованность нагнетателя 0.5% (РЕЗЕРВ)
	DI_03_R	(N_Pair:=6, DI_K0:= DI_K[2].RR.10,	DIb_K0:= DI_K[2].RR.11,			K_OUT:= kontroller.DIn_[4].val);
	// сигнал: Загазованность нагнетателя 1.0% (РЕЗЕРВ)		обрыв:  Загазованность нагнетателя 1.0% (РЕЗЕРВ)
	DI_03_R	(N_Pair:=7, DI_K0:= DI_K[2].RR.12,	DIb_K0:= DI_K[2].RR.13,			K_OUT:= kontroller.DIn_[4].val);
	// сигнал: Не подключено								обрыв: Не подключено
	DI_03_R	(N_Pair:=8, DI_K0:= 0,				DIb_K0:= 0,						K_OUT:= kontroller.DIn_[4].val);
	
	
	kontroller.DIn_[5].f		:= 5;	// .0 - есть в проекте		.1 - входные		.2 - достоверность		
	kontroller.DIn_[5].f.2		:= DI_K[3].VeraB;	// достоверность из драйвера RWH (=1 - достоверно)	
	//kontroller.DIn_[5].f.2		:= (kontroller.DIn_[0].val.1=0);		// недостоверность - получим их NodeErr модуля ???		
	//
	// сигнал: ПНС включен					обрыв:  ПНС включен
	DI_03_R	(N_Pair:=1, DI_K0:= DI_K[3].RR.0,	DIb_K0:= DI_K[3].RR.1,			K_OUT:= kontroller.DIn_[5].val);
	// сигнал: НУ1 включен					обрыв:  НУ1 включен
	DI_03_R	(N_Pair:=2, DI_K0:= DI_K[3].RR.2,	DIb_K0:= DI_K[3].RR.3,			K_OUT:= kontroller.DIn_[5].val);
	// сигнал: НУ2 включен				обрыв:  НУ2 включен
	DI_03_R	(N_Pair:=3, DI_K0:= DI_K[3].RR.4,	DIb_K0:= DI_K[3].RR.5,			K_OUT:= kontroller.DIn_[5].val);
	// сигнал: Вентилятор АВО масла №1 включен	обрыв:  Вентилятор АВО масла №1 включен
	DI_03_R	(N_Pair:=4, DI_K0:= DI_K[3].RR.6,	DIb_K0:= DI_K[3].RR.7,			K_OUT:= kontroller.DIn_[5].val);
	// сигнал: Вентилятор АВО масла №2 включен	обрыв:  Вентилятор АВО масла №2 включен
	DI_03_R	(N_Pair:=5, DI_K0:= DI_K[3].RR.8,	DIb_K0:= DI_K[3].RR.9,			K_OUT:= kontroller.DIn_[5].val);
	// сигнал: Вентилятор АВО масла №3 включен	обрыв:  Вентилятор АВО масла №3 включен
	DI_03_R	(N_Pair:=6, DI_K0:= DI_K[3].RR.10,	DIb_K0:= DI_K[3].RR.11,			K_OUT:= kontroller.DIn_[5].val);
	// сигнал: Вентилятор АВО масла №4 включен	обрыв:  Вентилятор АВО масла №4 включен
	DI_03_R	(N_Pair:=7, DI_K0:= DI_K[3].RR.12,	DIb_K0:= DI_K[3].RR.13,			K_OUT:= kontroller.DIn_[5].val);
	// сигнал: Не подключено					обрыв: Не подключено
	DI_03_R	(N_Pair:=8, DI_K0:= 0,				DIb_K0:= 0,						K_OUT:= kontroller.DIn_[5].val);
	

	kontroller.DIn_[6].f		:= 5;	// .0 - есть в проекте		.1 - входные		.2 - достоверность		
	kontroller.DIn_[6].f.2		:= DI_K[4].VeraB;	// достоверность из драйвера RWH (=1 - достоверно)	
	//kontroller.DIn_[6].f.2		:= (kontroller.DIn_[0].val.1=0);		// недостоверность - получим их NodeErr модуля ???		
	//
	// сигнал: Готовность возбудителя			обрыв:  Готовность возбудителя
	DI_03_R	(N_Pair:=1, DI_K0:= DI_K[4].RR.0,	DIb_K0:= DI_K[4].RR.1,			K_OUT:= kontroller.DIn_[6].val);
	// сигнал: Разрешение загрузки ГПА			обрыв:  Разрешение загрузки ГПА
	DI_03_R	(N_Pair:=2, DI_K0:= DI_K[4].RR.2,	DIb_K0:= DI_K[4].RR.3,			K_OUT:= kontroller.DIn_[6].val);
	// сигнал: Возбудитель неисправен			обрыв:  Возбудитель неисправен
	DI_03_R	(N_Pair:=3, DI_K0:= DI_K[4].RR.4,	DIb_K0:= DI_K[4].RR.5,			K_OUT:= kontroller.DIn_[6].val);
	// сигнал: Авария возбудителя				обрыв:  Авария возбудителя
	DI_03_R	(N_Pair:=4, DI_K0:= DI_K[4].RR.6,	DIb_K0:= DI_K[4].RR.7,			K_OUT:= kontroller.DIn_[6].val);
	// сигнал: Неисправность цепи управления АВР пит.возбудителя	обрыв:  Неисправность цепи управления АВР пит.возбудителя
	DI_03_R	(N_Pair:=5, DI_K0:= DI_K[4].RR.8,	DIb_K0:= DI_K[4].RR.9,			K_OUT:= kontroller.DIn_[6].val);
	// сигнал: Не подключено					обрыв: Не подключено
	DI_03_R	(N_Pair:=6, DI_K0:= 0,				DIb_K0:= 0,						K_OUT:= kontroller.DIn_[6].val);
	// сигнал: Не подключено					обрыв: Не подключено
	DI_03_R	(N_Pair:=7, DI_K0:= 0,				DIb_K0:= 0,						K_OUT:= kontroller.DIn_[6].val);
	// сигнал: Не подключено					обрыв: Не подключено
	DI_03_R	(N_Pair:=8, DI_K0:= 0,				DIb_K0:= 0,						K_OUT:= kontroller.DIn_[6].val);


	kontroller.DIn_[7].f		:= 5;	// .0 - есть в проекте		.1 - входные		.2 - достоверность		
	kontroller.DIn_[7].f.2		:= DI_K[5].VeraB;	// достоверность из драйвера RWH (=1 - достоверно)	
	//kontroller.DIn_[7].f.2		:= (kontroller.DIn_[0].val.1=0);		// недостоверность - получим их NodeErr модуля ???		
	//
	// сигнал: МВ включен						обрыв:  МВ включен
	DI_03_R	(N_Pair:=1, DI_K0:= DI_K[5].RR.0,	DIb_K0:= DI_K[5].RR.1,			K_OUT:= kontroller.DIn_[7].val);
	// сигнал: МВ отключен						обрыв:  МВ отключен
	DI_03_R	(N_Pair:=2, DI_K0:= DI_K[5].RR.2,	DIb_K0:= DI_K[5].RR.3,			K_OUT:= kontroller.DIn_[7].val);
	// сигнал: МВ в контр.положении (тележка выкачена)	обрыв:  МВ в контр.положении (тележка выкачена)
	DI_03_R	(N_Pair:=3, DI_K0:= DI_K[5].RR.4,	DIb_K0:= DI_K[5].RR.5,			K_OUT:= kontroller.DIn_[7].val);
	// сигнал: Пожар ГПА (РЕЗЕРВ)				обрыв:  Пожар ГПА (РЕЗЕРВ)
	DI_03_R	(N_Pair:=4, DI_K0:= DI_K[5].RR.6,	DIb_K0:= DI_K[5].RR.7,			K_OUT:= kontroller.DIn_[7].val);
	// сигнал: Наличие тока возбуждения (РЕЗЕРВ)	обрыв:  Наличие тока возбуждения (РЕЗЕРВ)
	DI_03_R	(N_Pair:=5, DI_K0:= DI_K[5].RR.8,	DIb_K0:= DI_K[5].RR.9,			K_OUT:= kontroller.DIn_[7].val);
	// сигнал: Неисправность КРУ (РЕЗЕРВ)		обрыв:  Неисправность КРУ (РЕЗЕРВ)		
	DI_03_R	(N_Pair:=6, DI_K0:= DI_K[5].RR.10,	DIb_K0:= DI_K[5].RR.11,			K_OUT:= kontroller.DIn_[7].val);
	// сигнал: Нет 10кВ (РЕЗЕРВ)				обрыв:  Нет 10кВ (РЕЗЕРВ)
	DI_03_R	(N_Pair:=7, DI_K0:= DI_K[5].RR.12,	DIb_K0:= DI_K[5].RR.13,			K_OUT:= kontroller.DIn_[7].val);
	// сигнал: Не подключено					обрыв: Не подключено
	DI_03_R	(N_Pair:=8, DI_K0:= 0,				DIb_K0:= 0,						K_OUT:= kontroller.DIn_[7].val);
	

	kontroller.DIn_[8].f		:= 5;	// .0 - есть в проекте		.1 - входные		.2 - достоверность		
	kontroller.DIn_[8].f.2		:= DI_K[6].VeraB;	// достоверность из драйвера RWH (=1 - достоверно)	
	//kontroller.DIn_[8].f.2		:= (kontroller.DIn_[0].val.1=0);		// недостоверность - получим их NodeErr модуля ???
	//
	// сигнал: Аварийное отключение выключателя		обрыв:  Аварийное отключение выключателя
	DI_03_R	(N_Pair:=1, DI_K0:= DI_K[6].RR.0,		DIb_K0:= DI_K[6].RR.1,			K_OUT:= kontroller.DIn_[8].val);
	// сигнал: Асинхронный ход, перегрузка			обрыв:  Асинхронный ход, перегрузка
	DI_03_R	(N_Pair:=2, DI_K0:= DI_K[6].RR.2,		DIb_K0:= DI_K[6].RR.3,			K_OUT:= kontroller.DIn_[8].val);
	// сигнал: Автомат ШУ в ячейке ГПА включен		обрыв:  Автомат ШУ в ячейке ГПА включен
	DI_03_R	(N_Pair:=3, DI_K0:= DI_K[6].RR.4,		DIb_K0:= DI_K[6].RR.5,			K_OUT:= kontroller.DIn_[8].val);
	// сигнал: Автомат ШП в ячейке ГПА включен		обрыв:  Автомат ШП в ячейке ГПА включен
	DI_03_R	(N_Pair:=4, DI_K0:= DI_K[6].RR.6,		DIb_K0:= DI_K[6].RR.7,			K_OUT:= kontroller.DIn_[8].val);
	// сигнал: Напряжение на секции в норме			обрыв:  Напряжение на секции в норме
	DI_03_R	(N_Pair:=5, DI_K0:= DI_K[6].RR.8,		DIb_K0:= DI_K[6].RR.9,			K_OUT:= kontroller.DIn_[8].val);
	// сигнал: Переключатель в положении "Реакторный пуск"	обрыв:  Переключатель в положении "Реакторный пуск"
	DI_03_R	(N_Pair:=6, DI_K0:= DI_K[6].RR.10,		DIb_K0:= DI_K[6].RR.11,			K_OUT:= kontroller.DIn_[8].val);
	// сигнал: Не подключено						обрыв: Не подключено
	DI_03_R	(N_Pair:=7, DI_K0:= 0,					DIb_K0:= 0,						K_OUT:= kontroller.DIn_[8].val);
	// сигнал: Не подключено						обрыв: Не подключено
	DI_03_R	(N_Pair:=8, DI_K0:= 0,					DIb_K0:= 0,						K_OUT:= kontroller.DIn_[8].val);

	
	kontroller.DIn_[9].f		:= 5;	// .0 - есть в проекте		.1 - входные		.2 - достоверность		
	kontroller.DIn_[9].f.2		:= DI_K[7].VeraB;	// достоверность из драйвера RWH (=1 - достоверно)	
	//kontroller.DIn_[9].f.2		:= (kontroller.DIn_[0].val.1=0);		// недостоверность - получим их NodeErr модуля ???		
	//
	// сигнал: Частотный пуск						обрыв:  Частотный пуск
	DI_03_R	(N_Pair:=1, DI_K0:= DI_K[7].RR.0,		DIb_K0:= DI_K[7].RR.1,			K_OUT:= kontroller.DIn_[9].val);
	// сигнал: Неуспешный частотный пуск			обрыв:  Неуспешный частотный пуск
	DI_03_R	(N_Pair:=2, DI_K0:= DI_K[7].RR.2,		DIb_K0:= DI_K[7].RR.3,			K_OUT:= kontroller.DIn_[9].val);
	// сигнал: Режим ручного регулирования			обрыв:  Режим ручного регулирования
	DI_03_R	(N_Pair:=3, DI_K0:= DI_K[7].RR.4,		DIb_K0:= DI_K[7].RR.5,			K_OUT:= kontroller.DIn_[9].val);
	// сигнал: АО КЦ (от ШКС)						обрыв:  АО КЦ (от ШКС)
	DI_03_R	(N_Pair:=4, DI_K0:= DI_K[7].RR.6,		DIb_K0:= DI_K[7].RR.7,			K_OUT:= kontroller.DIn_[9].val);
	// сигнал: НО ГПА (от кнопки ШУ ЭГПА)			обрыв:  НО ГПА (от кнопки ШУ ЭГПА)
	DI_03_R	(N_Pair:=5, DI_K0:= DI_K[7].RR.8,		DIb_K0:= DI_K[7].RR.9,			K_OUT:= kontroller.DIn_[9].val);
	// сигнал: АО ГПА (от кнопки ШУ ЭГПА)			обрыв:  АО ГПА (от кнопки ШУ ЭГПА)				
	DI_03_R	(N_Pair:=6, DI_K0:= DI_K[7].RR.10,		DIb_K0:= DI_K[7].RR.11,			K_OUT:= kontroller.DIn_[9].val);
	// сигнал: АО ГПА (от кнопки на ПРУ ЭГПА)		обрыв:  АО ГПА (от кнопки на ПРУ ЭГПА)
	DI_03_R	(N_Pair:=7, DI_K0:= DI_K[7].RR.12,		DIb_K0:= DI_K[7].RR.13,			K_OUT:= kontroller.DIn_[9].val);
	// сигнал: Не подключено						обрыв: Не подключено
	DI_03_R	(N_Pair:=8, DI_K0:= 0,					DIb_K0:= 0,						K_OUT:= kontroller.DIn_[9].val);

	
	kontroller.DIn_[10].f		:= 5;	// .0 - есть в проекте		.1 - входные		.2 - достоверность		
	kontroller.DIn_[10].f.2		:= DI_K[8].VeraB;	// достоверность из драйвера RWH (=1 - достоверно)	
	//kontroller.DIn_[10].f.2		:= (kontroller.DIn_[0].val.1=0);		// недостоверность - получим их NodeErr модуля ???		
	//
	// сигнал: ТЭН МБ включен						обрыв:  ТЭН МБ включен
	DI_03_R	(N_Pair:=1, DI_K0:= DI_K[8].RR.0,		DIb_K0:= DI_K[8].RR.1,			K_OUT:= kontroller.DIn_[10].val);
	// сигнал: ТЭН колл. включен					обрыв:  ТЭН колл. включен
	DI_03_R	(N_Pair:=2, DI_K0:= DI_K[8].RR.2,		DIb_K0:= DI_K[8].RR.3,			K_OUT:= kontroller.DIn_[10].val);
	// сигнал: Калорифер АВО масла включен			обрыв:  Калорифер АВО масла включен
	DI_03_R	(N_Pair:=3, DI_K0:= DI_K[8].RR.4,		DIb_K0:= DI_K[8].RR.5,			K_OUT:= kontroller.DIn_[10].val);
	// сигнал: Насос циркуляции масла включен		обрыв:  Насос циркуляции масла включен
	DI_03_R	(N_Pair:=4, DI_K0:= DI_K[8].RR.6,		DIb_K0:= DI_K[8].RR.7,			K_OUT:= kontroller.DIn_[10].val);
	// сигнал: НКУ ГПА ввод 1 включен				обрыв:  НКУ ГПА ввод 1 включен
	DI_03_R	(N_Pair:=5, DI_K0:= DI_K[8].RR.8,		DIb_K0:= DI_K[8].RR.9,			K_OUT:= kontroller.DIn_[10].val);
	// сигнал: НКУ ГПА ввод 2 включен				обрыв:  НКУ ГПА ввод 2 включен
	DI_03_R	(N_Pair:=6, DI_K0:= DI_K[8].RR.10,		DIb_K0:= DI_K[8].RR.11,			K_OUT:= kontroller.DIn_[10].val);
	// сигнал: Не подключено						обрыв: Не подключено
	DI_03_R	(N_Pair:=7, DI_K0:= 0,					DIb_K0:= 0,						K_OUT:= kontroller.DIn_[10].val);
	// сигнал: Не подключено						обрыв: Не подключено
	DI_03_R	(N_Pair:=8, DI_K0:= 0,					DIb_K0:= 0,						K_OUT:= kontroller.DIn_[10].val);

	
	kontroller.DIn_[11].f		:= 5;	// .0 - есть в проекте		.1 - входные		.2 - достоверность		
	kontroller.DIn_[11].f.2		:= DI_K[9].VeraB;	// достоверность из драйвера RWH (=1 - достоверно)	
	//kontroller.DIn_[11].f.2		:= (kontroller.DIn_[0].val.1=0);		// недостоверность - получим их NodeErr модуля ???		
	//
	//	сигнал: Неисправность =24В, U1.1 (Пит.контроллера 1, Х1)	обрыв: Нет обрыва
	DI_03_R	(N_Pair:=1, DI_K0:= DI_K[9].RR.0,						DIb_K0:= 1,			K_OUT:= kontroller.DIn_[11].val);
	// сигнал: Неисправность =24В, U1.2 (Пит.контроллера 2, Х2)		обрыв: Нет обрыва
	DI_03_R	(N_Pair:=2, DI_K0:= DI_K[9].RR.1,						DIb_K0:= 1,			K_OUT:= kontroller.DIn_[11].val);
	// сигнал: Неисправность БП3 (=24В, Пит.внутр.цепей)			обрыв: Нет обрыва
	DI_03_R	(N_Pair:=3, DI_K0:= DI_K[9].RR.2,						DIb_K0:= 1,			K_OUT:= kontroller.DIn_[11].val);
	// сигнал: Неисправность БП4 (=24В, Пит.внутр.цепей)			обрыв: Нет обрыва	
	DI_03_R	(N_Pair:=4, DI_K0:= DI_K[9].RR.3,						DIb_K0:= 1,			K_OUT:= kontroller.DIn_[11].val);
	// сигнал: Неисправность БП5 (=24В, Пит.вх.дискр.сигналов)		обрыв: Нет обрыва	
	DI_03_R	(N_Pair:=5, DI_K0:= DI_K[9].RR.4,						DIb_K0:= 1,			K_OUT:= kontroller.DIn_[11].val);
	// сигнал: Неисправность БП6 (=24В, Пит.вх.дискр.сигналов)		обрыв: Нет обрыва	
	DI_03_R	(N_Pair:=6, DI_K0:= DI_K[9].RR.5,						DIb_K0:= 1,			K_OUT:= kontroller.DIn_[11].val);
	// сигнал: Неисправность БП7 и БП8 (=24В, Пит.кранов)			обрыв: Нет обрыва
	DI_03_R	(N_Pair:=7, DI_K0:= DI_K[9].RR.6,						DIb_K0:= 1,			K_OUT:= kontroller.DIn_[11].val);
	// сигнал: Неисправность БП9 и БП10 (=24В, Рез.)				обрыв: Нет обрыва
	DI_03_R	(N_Pair:=8, DI_K0:= DI_K[9].RR.7,						DIb_K0:= 1,			K_OUT:= kontroller.DIn_[11].val);
	
	
	kontroller.DIn_[12].f		:= 5;	// .0 - есть в проекте		.1 - входные		.2 - достоверность		
	kontroller.DIn_[12].f.2		:= DI_K[9].VeraB;	// достоверность из драйвера RWH (=1 - достоверно)	
	//kontroller.DIn_[12].f.2		:= (kontroller.DIn_[0].val.1=0);		// недостоверность - получим их NodeErr модуля ???		
	//
	// сигнал: Нет обрыва цепи управления МВ			обрыв: Нет обрыва
	DI_03_R	(N_Pair:=1, DI_K0:= DI_K[9].RR.8,			DIb_K0:= 1,			K_OUT:= kontroller.DIn_[12].val);
	// сигнал: Контроль =220В БРЭО						обрыв: Нет обрыва	
	DI_03_R	(N_Pair:=2, DI_K0:= DI_K[9].RR.9,			DIb_K0:= 1,			K_OUT:= kontroller.DIn_[12].val);
	// сигнал: Нет питания (~220В)						обрыв: Нет обрыва	
	DI_03_R	(N_Pair:=3, DI_K0:= DI_K[9].RR.10,			DIb_K0:= 1,			K_OUT:= kontroller.DIn_[12].val);
	// сигнал: Нет питания (=220В)						обрыв: Нет обрыва	
	DI_03_R	(N_Pair:=4, DI_K0:= DI_K[9].RR.11,			DIb_K0:= 1,			K_OUT:= kontroller.DIn_[12].val);
	// сигнал: Неисправность БП11 (=24В, Пит.МПУ)		обрыв: Нет обрыва
	DI_03_R	(N_Pair:=5, DI_K0:= DI_K[9].RR.12,			DIb_K0:= 1,			K_OUT:= kontroller.DIn_[12].val);
	// сигнал: Неисправность БП12 (=24В, Пит.МПУ)		обрыв: Нет обрыва
	DI_03_R	(N_Pair:=6, DI_K0:= DI_K[9].RR.13,			DIb_K0:= 1,			K_OUT:= kontroller.DIn_[12].val);
	// сигнал: Не подключено							обрыв: Не подключено
	DI_03_R	(N_Pair:=7, DI_K0:= 0,						DIb_K0:= 0,			K_OUT:= kontroller.DIn_[12].val);
	// сигнал: Не подключено							обрыв: Не подключено	
	DI_03_R	(N_Pair:=8, DI_K0:= 0,						DIb_K0:= 0,			K_OUT:= kontroller.DIn_[12].val);
	

	kontroller.DIn_[13].f		:= 5;	// .0 - есть в проекте		.1 - входные		.2 - достоверность		
	kontroller.DIn_[13].f.2		:= DI_K[10].VeraB;	// достоверность из драйвера RWH (=1 - достоверно)	
	//kontroller.DIn_[13].f.2		:= (kontroller.DIn_[0].val.1=0);		// недостоверность - получим их NodeErr модуля ???		
	//
	// сигнал: Дверь ШУ САУ открыта (дискрет.сторона)			обрыв: Нет обрыва	
	DI_03_R	(N_Pair:=1, DI_K0:= DI_K[10].RR.0,					DIb_K0:= 1,			K_OUT:= kontroller.DIn_[13].val);
	// сигнал: Дверь ШУ САУ открыта (аналог.сторона)			обрыв: Нет обрыва	
	DI_03_R	(N_Pair:=2, DI_K0:= DI_K[10].RR.1,					DIb_K0:= 1,			K_OUT:= kontroller.DIn_[13].val);
	// сигнал: Не подключено									обрыв: Не подключено
	DI_03_R	(N_Pair:=3, DI_K0:= 0,								DIb_K0:= 0,			K_OUT:= kontroller.DIn_[13].val);
	// сигнал: Не подключено									обрыв: Не подключено
	DI_03_R	(N_Pair:=4, DI_K0:= 0,								DIb_K0:= 0,			K_OUT:= kontroller.DIn_[13].val);
	// сигнал: Не подключено									обрыв: Не подключено
	DI_03_R	(N_Pair:=5, DI_K0:= 0,								DIb_K0:= 0,			K_OUT:= kontroller.DIn_[13].val);
	// сигнал: Не подключено									обрыв: Не подключено
	DI_03_R	(N_Pair:=6, DI_K0:= 0,								DIb_K0:= 0,			K_OUT:= kontroller.DIn_[13].val);
	// сигнал: ЩАВР ввод №1 в работе							обрыв: Нет обрыва
	DI_03_R	(N_Pair:=7, DI_K0:= DI_K[10].RR.6,					DIb_K0:= 1,			K_OUT:= kontroller.DIn_[13].val);
	// сигнал: ЩАВР ввод №2 в работе							обрыв: Нет обрыва
	DI_03_R	(N_Pair:=8, DI_K0:= DI_K[10].RR.7,					DIb_K0:= 1,			K_OUT:= kontroller.DIn_[13].val);
	

	kontroller.DIn_[14].f		:= 5;	// .0 - есть в проекте		.1 - входные		.2 - достоверность		
	kontroller.DIn_[14].f.2		:= DI_K[10].VeraB;	// достоверность из драйвера RWH (=1 - достоверно)	
	//kontroller.DIn_[14].f.2		:= (kontroller.DIn_[0].val.1=0);		// недостоверность - получим их NodeErr модуля ???		
	//
	// сигнал: ЭО ГПА (от кнопки на ШУ ЭГПА)			обрыв: Нет обрыва
	DI_03_R	(N_Pair:=1, DI_K0:= DI_K[10].RR.8,			DIb_K0:= 1,			K_OUT:= kontroller.DIn_[14].val);
	// сигнал: ЭО ГПА (от кнопки на ПРУ ЭГПА)			обрыв: Нет обрыва
	DI_03_R	(N_Pair:=2, DI_K0:= DI_K[10].RR.9,			DIb_K0:= 1,			K_OUT:= kontroller.DIn_[14].val);
	// сигнал: Наличие напряжения на ПНС				обрыв: Нет обрыва
	DI_03_R	(N_Pair:=3, DI_K0:= DI_K[10].RR.10,			DIb_K0:= 1,			K_OUT:= kontroller.DIn_[14].val);
	// сигнал: Наличие напряжения на НУ1				обрыв: Нет обрыва	
	DI_03_R	(N_Pair:=4, DI_K0:= DI_K[10].RR.11,			DIb_K0:= 1,			K_OUT:= kontroller.DIn_[14].val);
	// сигнал: Наличие напряжения на НУ2				обрыв: Нет обрыва	
	DI_03_R	(N_Pair:=5, DI_K0:= DI_K[10].RR.12,			DIb_K0:= 1,			K_OUT:= kontroller.DIn_[14].val);
	// сигнал: Наличие напряжения на ЦМН подано			обрыв: Нет обрыва	
	DI_03_R	(N_Pair:=6, DI_K0:= DI_K[10].RR.13,			DIb_K0:= 1,			K_OUT:= kontroller.DIn_[14].val);
	// сигнал: Не подключено							обрыв: Не подключено
	DI_03_R	(N_Pair:=7, DI_K0:= 0,						DIb_K0:= 0,			K_OUT:= kontroller.DIn_[14].val);
	// сигнал: Не подключено							обрыв: Не подключено
	DI_03_R	(N_Pair:=8, DI_K0:= 0,						DIb_K0:= 0,			K_OUT:= kontroller.DIn_[14].val);
	
	
	kontroller.DIn_[15].f		:= 5;	// .0 - есть в проекте		.1 - входные		.2 - достоверность		
	kontroller.DIn_[15].f.2		:= DI_K[11].VeraB;	// достоверность из драйвера RWH (=1 - достоверно)	
	//kontroller.DIn_[15].f.2		:= (kontroller.DIn_[0].val.1=0);		// недостоверность - получим их NodeErr модуля ???		
	//
	// сигнал: Не подключено				обрыв: Не подключено
	DI_03_R	(N_Pair:=1, DI_K0:= 0,			DIb_K0:= 0,			K_OUT:= kontroller.DIn_[15].val);
	// сигнал: Не подключено				обрыв: Не подключено
	DI_03_R	(N_Pair:=2, DI_K0:= 0,			DIb_K0:= 0,			K_OUT:= kontroller.DIn_[15].val);
	// сигнал: Не подключено				обрыв: Не подключено
	DI_03_R	(N_Pair:=3, DI_K0:= 0,			DIb_K0:= 0,			K_OUT:= kontroller.DIn_[15].val);
	// сигнал: Не подключено				обрыв: Не подключено
	DI_03_R	(N_Pair:=4, DI_K0:= 0,			DIb_K0:= 0,			K_OUT:= kontroller.DIn_[15].val);
	// сигнал: Не подключено				обрыв: Не подключено
	DI_03_R	(N_Pair:=5, DI_K0:= 0,			DIb_K0:= 0,			K_OUT:= kontroller.DIn_[15].val);
	// сигнал: Не подключено				обрыв: Не подключено
	DI_03_R	(N_Pair:=6, DI_K0:= 0,			DIb_K0:= 0,			K_OUT:= kontroller.DIn_[15].val);
	// сигнал: Не подключено				обрыв: Не подключено
	DI_03_R	(N_Pair:=7, DI_K0:= 0,			DIb_K0:= 0,			K_OUT:= kontroller.DIn_[15].val);
	// сигнал: Не подключено				обрыв: Не подключено
	DI_03_R	(N_Pair:=8, DI_K0:= 0,			DIb_K0:= 0,			K_OUT:= kontroller.DIn_[15].val);

	
	kontroller.DIn_[16].f		:= 5;	// .0 - есть в проекте		.1 - входные		.2 - достоверность		
	kontroller.DIn_[16].f.2		:= DI_K[12].VeraB;	// достоверность из драйвера RWH (=1 - достоверно)	
	//kontroller.DIn_[16].f.2		:= (kontroller.DIn_[0].val.1=0);		// недостоверность - получим их NodeErr модуля ???		
	//
	// сигнал: Кран 1 обрыв СО						обрыв: Нет обрыва	
	DI_03_R	(N_Pair:=1, DI_K0:= DI_K[12].RR.0,		DIb_K0:= 1,			K_OUT:= kontroller.DIn_[16].val);
	// сигнал: Кран 1 обрыв СЗ						обрыв: Нет обрыва	
	DI_03_R	(N_Pair:=2, DI_K0:= DI_K[12].RR.1,		DIb_K0:= 1,			K_OUT:= kontroller.DIn_[16].val);
	// сигнал: Кран 2 обрыв СО						обрыв: Нет обрыва	
	DI_03_R	(N_Pair:=3, DI_K0:= DI_K[12].RR.2,		DIb_K0:= 1,			K_OUT:= kontroller.DIn_[16].val);
	// сигнал: Кран 2 обрыв СЗ						обрыв: Нет обрыва	
	DI_03_R	(N_Pair:=4, DI_K0:= DI_K[12].RR.3,		DIb_K0:= 1,			K_OUT:= kontroller.DIn_[16].val);
	// сигнал: Кран 3 обрыв СО						обрыв: Нет обрыва	
	DI_03_R	(N_Pair:=5, DI_K0:= DI_K[12].RR.4,		DIb_K0:= 1,			K_OUT:= kontroller.DIn_[16].val);
	// сигнал: Кран 3 обрыв СЗ						обрыв: Нет обрыва	
	DI_03_R	(N_Pair:=6, DI_K0:= DI_K[12].RR.5,		DIb_K0:= 1,			K_OUT:= kontroller.DIn_[16].val);
	// сигнал: Кран 3b обрыв СО						обрыв: Нет обрыва	
	DI_03_R	(N_Pair:=7, DI_K0:= DI_K[12].RR.6,		DIb_K0:= 1,			K_OUT:= kontroller.DIn_[16].val);
	// сигнал: Кран 3b обрыв СЗ						обрыв: Нет обрыва	
	DI_03_R	(N_Pair:=8, DI_K0:= DI_K[12].RR.7,		DIb_K0:= 1,			K_OUT:= kontroller.DIn_[16].val);

	
	kontroller.DIn_[17].f		:= 5;	// .0 - есть в проекте		.1 - входные		.2 - достоверность		
	kontroller.DIn_[17].f.2		:= DI_K[12].VeraB;	// достоверность из драйвера RWH (=1 - достоверно)	
	//kontroller.DIn_[17].f.2		:= (kontroller.DIn_[0].val.1=0);		// недостоверность - получим их NodeErr модуля ???		
	//
	// сигнал: Кран 4 обрыв СО						обрыв: Нет обрыва
	DI_03_R	(N_Pair:=1, DI_K0:= DI_K[12].RR.8,		DIb_K0:= 1,			K_OUT:= kontroller.DIn_[17].val);
	// сигнал: Кран 4 обрыв СЗ						обрыв: Нет обрыва
	DI_03_R	(N_Pair:=2, DI_K0:= DI_K[12].RR.9,		DIb_K0:= 1,			K_OUT:= kontroller.DIn_[17].val);
	// сигнал: Кран 5 обрыв СО						обрыв: Нет обрыва
	DI_03_R	(N_Pair:=3, DI_K0:= DI_K[12].RR.10,		DIb_K0:= 1,			K_OUT:= kontroller.DIn_[17].val);
	// сигнал: Кран 5 обрыв СЗ						обрыв: Нет обрыва
	DI_03_R	(N_Pair:=4, DI_K0:= DI_K[12].RR.11,		DIb_K0:= 1,			K_OUT:= kontroller.DIn_[17].val);
	// сигнал: Кран 6 обрыв СО						обрыв: Нет обрыва
	DI_03_R	(N_Pair:=5, DI_K0:= DI_K[12].RR.12,		DIb_K0:= 1,			K_OUT:= kontroller.DIn_[17].val);
	// сигнал: Кран 6 обрыв СЗ						обрыв: Нет обрыва
	DI_03_R	(N_Pair:=6, DI_K0:= DI_K[12].RR.13,		DIb_K0:= 1,			K_OUT:= kontroller.DIn_[17].val);
	// сигнал: Не подключено						обрыв: Не подключено
	DI_03_R	(N_Pair:=7, DI_K0:= 0,					DIb_K0:= 0,			K_OUT:= kontroller.DIn_[17].val);
	// сигнал: Не подключено						обрыв: Не подключено
	DI_03_R	(N_Pair:=8, DI_K0:= 0,					DIb_K0:= 0,			K_OUT:= kontroller.DIn_[17].val);
	

	kontroller.DIn_[18].f		:= 5;	// .0 - есть в проекте		.1 - входные		.2 - достоверность		
	kontroller.DIn_[18].f.2		:= DI_K[13].VeraB;	// достоверность из драйвера RWH (=1 - достоверно)	
	//kontroller.DIn_[18].f.2		:= (kontroller.DIn_[0].val.1=0);		// недостоверность - получим их NodeErr модуля ???		
	//
	// сигнал: Поток масла после АВОм > 85 л/м						обрыв: Нет обрыва
	DI_03_R	(N_Pair:=1, DI_K0:= DI_K[13].RR.0,		DIb_K0:= 1,			K_OUT:= kontroller.DIn_[18].val);
	// сигнал: Не подключено						обрыв: Не подключено
	DI_03_R	(N_Pair:=2, DI_K0:= DI_K[13].RR.1,		DIb_K0:= 1,			K_OUT:= kontroller.DIn_[18].val);
	// сигнал: Не подключено						обрыв: Не подключено
	DI_03_R	(N_Pair:=3, DI_K0:= 0,					DIb_K0:= 0,			K_OUT:= kontroller.DIn_[18].val);
	// сигнал: Не подключено						обрыв: Не подключено
	DI_03_R	(N_Pair:=4, DI_K0:= 0,					DIb_K0:= 0,			K_OUT:= kontroller.DIn_[18].val);
	// сигнал: Не подключено						обрыв: Не подключено
	DI_03_R	(N_Pair:=5, DI_K0:= 0,					DIb_K0:= 0,			K_OUT:= kontroller.DIn_[18].val);
	// сигнал: Не подключено						обрыв: Не подключено
	DI_03_R	(N_Pair:=6, DI_K0:= 0,					DIb_K0:= 0,			K_OUT:= kontroller.DIn_[18].val);
	// сигнал: Не подключено						обрыв: Не подключено
	DI_03_R	(N_Pair:=7, DI_K0:= 0,					DIb_K0:= 0,			K_OUT:= kontroller.DIn_[18].val);
	// сигнал: Не подключено						обрыв: Не подключено
	DI_03_R	(N_Pair:=8, DI_K0:= 0,					DIb_K0:= 0,			K_OUT:= kontroller.DIn_[18].val);
	
	
	kontroller.DIn_[19].f		:= 5;	// .0 - есть в проекте		.1 - входные		.2 - достоверность		
	kontroller.DIn_[19].f.2		:= DI_K[13].VeraB;	// достоверность из драйвера RWH (=1 - достоверно)	
	//kontroller.DIn_[19].f.2		:= (kontroller.DIn_[0].val.1=0);		// недостоверность - получим их NodeErr модуля ???		
	// сигнал: Не подключено						обрыв: Не подключено
	DI_03_R	(N_Pair:=1, DI_K0:= 0,					DIb_K0:= 0,			K_OUT:= kontroller.DIn_[19].val);
	// сигнал: Не подключено						обрыв: Не подключено
	DI_03_R	(N_Pair:=2, DI_K0:= 0,					DIb_K0:= 0,			K_OUT:= kontroller.DIn_[19].val);
	// сигнал: Не подключено						обрыв: Не подключено
	DI_03_R	(N_Pair:=3, DI_K0:= 0,					DIb_K0:= 0,			K_OUT:= kontroller.DIn_[19].val);
	// сигнал: Не подключено						обрыв: Не подключено
	DI_03_R	(N_Pair:=4, DI_K0:= 0,					DIb_K0:= 0,			K_OUT:= kontroller.DIn_[19].val);
	// сигнал: Не подключено						обрыв: Не подключено
	DI_03_R	(N_Pair:=5, DI_K0:= 0,					DIb_K0:= 0,			K_OUT:= kontroller.DIn_[19].val);
	// сигнал: Не подключено						обрыв: Не подключено
	DI_03_R	(N_Pair:=6, DI_K0:= 0,					DIb_K0:= 0,			K_OUT:= kontroller.DIn_[19].val);
	// сигнал: Не подключено						обрыв: Не подключено
	DI_03_R	(N_Pair:=7, DI_K0:= 0,					DIb_K0:= 0,			K_OUT:= kontroller.DIn_[19].val);
	// сигнал: Не подключено						обрыв: Не подключено
	DI_03_R	(N_Pair:=8, DI_K0:= 0,					DIb_K0:= 0,			K_OUT:= kontroller.DIn_[19].val);
	
	///	
	//	Аварийное УСО поз.8
	///	
	kontroller.DIn_[20].f		:= 5;	// .0 - есть в проекте		.1 - входные		.2 - достоверность		
	kontroller.DIn_[20].f.2		:= DI_K[14].VeraB;	// достоверность из драйвера RWH (=1 - достоверно)	
	//kontroller.DIn_[20].f.2		:= (kontroller.DIn_[0].val.1=0);		// недостоверность - получим их NodeErr модуля ???		
	//
	// сигнал: АО цеха (от ШКС-04М)						обрыв: Нет обрыва
	DI_03_R	(N_Pair:=1, DI_K0:= DI_K[14].RR.0,		DIb_K0:= 1,			K_OUT:= kontroller.DIn_[20].val);
	// сигнал: Не подключено							обрыв: Не подключено
	DI_03_R	(N_Pair:=2, DI_K0:= 0,					DIb_K0:= 0,			K_OUT:= kontroller.DIn_[20].val);
	// сигнал: Не подключено							обрыв: Не подключено
	DI_03_R	(N_Pair:=3, DI_K0:= 0,					DIb_K0:= 0,			K_OUT:= kontroller.DIn_[20].val);
	// сигнал: МВ отключен								обрыв: Нет обрыва
	DI_03_R	(N_Pair:=4, DI_K0:= DI_K[14].RR.3,		DIb_K0:= 1,			K_OUT:= kontroller.DIn_[20].val);
	// сигнал: Кран 1 открыт							обрыв: Нет обрыва
	DI_03_R	(N_Pair:=5, DI_K0:= DI_K[14].RR.4,		DIb_K0:= 1,			K_OUT:= kontroller.DIn_[20].val);
	// сигнал: Кран 1 закрыт							обрыв: Нет обрыва
	DI_03_R	(N_Pair:=6, DI_K0:= DI_K[14].RR.5,		DIb_K0:= 1,			K_OUT:= kontroller.DIn_[20].val);
	// сигнал: Перепад давления масло-газ < 100 кПа		обрыв: Нет обрыва
	DI_03_R	(N_Pair:=7, DI_K0:= DI_K[14].RR.6,		DIb_K0:= 1,			K_OUT:= kontroller.DIn_[20].val);
	// сигнал: Кран 2 открыт							обрыв: Нет обрыва
	DI_03_R	(N_Pair:=8, DI_K0:= DI_K[14].RR.7,		DIb_K0:= 1,			K_OUT:= kontroller.DIn_[20].val);
	

	kontroller.DIn_[21].f		:= 5;	// .0 - есть в проекте		.1 - входные		.2 - достоверность		
	kontroller.DIn_[21].f.2		:= DI_K[14].VeraB;	// достоверность из драйвера RWH (=1 - достоверно)	
	//kontroller.DIn_[21].f.2		:= (kontroller.DIn_[0].val.1=0);		// недостоверность - получим их NodeErr модуля ???		
	//
	// сигнал: Кран 2 закрыт						обрыв: Нет обрыва
	DI_03_R	(N_Pair:=1, DI_K0:= DI_K[14].RR.8,		DIb_K0:= 1,			K_OUT:= kontroller.DIn_[21].val);
	// сигнал: НО ГПА (от кнопки на ШУ ЭГПА)		обрыв: Нет обрыва
	DI_03_R	(N_Pair:=2, DI_K0:= DI_K[14].RR.9,		DIb_K0:= 1,			K_OUT:= kontroller.DIn_[21].val);
	// сигнал: АО ГПА (от кнопки на ШУ ЭГПА)		обрыв: Нет обрыва
	DI_03_R	(N_Pair:=3, DI_K0:= DI_K[14].RR.10,		DIb_K0:= 1,			K_OUT:= kontroller.DIn_[21].val);
	// сигнал: АО ГПА (от кнопки на ПРУ ЭГПА)		обрыв: Нет обрыва
	DI_03_R	(N_Pair:=4, DI_K0:= DI_K[14].RR.11,		DIb_K0:= 1,			K_OUT:= kontroller.DIn_[21].val);
	// сигнал: Меандр активности К1/К2				обрыв: Нет обрыва
	DI_03_R	(N_Pair:=5, DI_K0:= DI_K[14].RR.12,		DIb_K0:= 1,			K_OUT:= kontroller.DIn_[21].val);
	// сигнал: Команда стать пассивным от К1/К2		обрыв: Нет обрыва
	DI_03_R	(N_Pair:=6, DI_K0:= DI_K[14].RR.13,		DIb_K0:= 1,			K_OUT:= kontroller.DIn_[21].val);
	// сигнал: Разрешить условный переход от К1/К2	обрыв: Нет обрыва
	DI_03_R	(N_Pair:=7, DI_K0:= DI_K[14].RR.14,		DIb_K0:= 1,			K_OUT:= kontroller.DIn_[21].val);
	// сигнал: Возбудитель неисправен				обрыв: Нет обрыва	
	DI_03_R	(N_Pair:=8, DI_K0:= DI_K[14].RR.15,		DIb_K0:= 1,			K_OUT:= kontroller.DIn_[21].val);
	
	///	
	//	Аварийное УСО поз.10
	///	
	kontroller.DIn_[22].f		:= 5;	// .0 - есть в проекте		.1 - входные		.2 - достоверность		
	kontroller.DIn_[22].f.2		:= DI_K[15].VeraB;	// достоверность из драйвера RWH (=1 - достоверно)	
	//kontroller.DIn_[22].f.2		:= (kontroller.DIn_[0].val.1=0);		// недостоверность - получим их NodeErr модуля ???		
	//
	// сигнал: Загазованность двигателя 1% (РЕЗЕРВ)		обрыв: Нет обрыва
	DI_03_R	(N_Pair:=1, DI_K0:= DI_K[15].RR.0,			DIb_K0:= 1,			K_OUT:= kontroller.DIn_[22].val);
	// сигнал: Загазованность нагнетателя 1% (РЕЗЕРВ)	обрыв: Нет обрыва
	DI_03_R	(N_Pair:=2, DI_K0:= DI_K[15].RR.1,			DIb_K0:= 1,			K_OUT:= kontroller.DIn_[22].val);
	// сигнал: Пожар ГПА								обрыв: Нет обрыва
	DI_03_R	(N_Pair:=3, DI_K0:= DI_K[15].RR.2,			DIb_K0:= 1,			K_OUT:= kontroller.DIn_[22].val);
	// сигнал: Не подключено							обрыв: Не подключено
	DI_03_R	(N_Pair:=4, DI_K0:= 0,						DIb_K0:= 0,			K_OUT:= kontroller.DIn_[22].val);
	// сигнал: Не подключено							обрыв: Не подключено
	DI_03_R	(N_Pair:=5, DI_K0:= 0,						DIb_K0:= 0,			K_OUT:= kontroller.DIn_[22].val);
	// сигнал: Не подключено							обрыв: Не подключено
	DI_03_R	(N_Pair:=6, DI_K0:= 0,						DIb_K0:= 0,			K_OUT:= kontroller.DIn_[22].val);
	// сигнал: Не подключено							обрыв: Не подключено
	DI_03_R	(N_Pair:=7, DI_K0:= 0,						DIb_K0:= 0,			K_OUT:= kontroller.DIn_[22].val);
	// сигнал: Не подключено							обрыв: Не подключено
	DI_03_R	(N_Pair:=8, DI_K0:= 0,						DIb_K0:= 0,			K_OUT:= kontroller.DIn_[22].val);

	
	kontroller.DIn_[23].f		:= 5;	// .0 - есть в проекте		.1 - входные		.2 - достоверность		
	kontroller.DIn_[23].f.2		:= DI_K[15].VeraB;	// достоверность из драйвера RWH (=1 - достоверно)	
	//kontroller.DIn_[23].f.2		:= (kontroller.DIn_[0].val.1=0);		// недостоверность - получим их NodeErr модуля ???		
	//
	// сигнал: Не подключено							обрыв: Не подключено
	DI_03_R	(N_Pair:=1, DI_K0:= 0,						DIb_K0:= 0,			K_OUT:= kontroller.DIn_[23].val);
	// сигнал: Не подключено							обрыв: Не подключено
	DI_03_R	(N_Pair:=2, DI_K0:= 0,						DIb_K0:= 0,			K_OUT:= kontroller.DIn_[23].val);
	// сигнал: Не подключено							обрыв: Не подключено
	DI_03_R	(N_Pair:=3, DI_K0:= 0,						DIb_K0:= 0,			K_OUT:= kontroller.DIn_[23].val);
	// сигнал: Не подключено							обрыв: Не подключено
	DI_03_R	(N_Pair:=4, DI_K0:= 0,						DIb_K0:= 0,			K_OUT:= kontroller.DIn_[23].val);
	// сигнал: Не подключено							обрыв: Не подключено
	DI_03_R	(N_Pair:=5, DI_K0:= 0,						DIb_K0:= 0,			K_OUT:= kontroller.DIn_[23].val);
	// сигнал: Не подключено							обрыв: Не подключено
	DI_03_R	(N_Pair:=6, DI_K0:= 0,						DIb_K0:= 0,			K_OUT:= kontroller.DIn_[23].val);
	// сигнал: Не подключено							обрыв: Не подключено
	DI_03_R	(N_Pair:=7, DI_K0:= 0,						DIb_K0:= 0,			K_OUT:= kontroller.DIn_[23].val);
	// сигнал: Не подключено							обрыв: Не подключено
	DI_03_R	(N_Pair:=8, DI_K0:= 0,						DIb_K0:= 0,			K_OUT:= kontroller.DIn_[23].val);

	
	
//////////////////////АНАЛОГОВЫЕ/////////////ПОЗ 15/////////////////МАЦП-16///////////////////////////////////////////////////

	// сигнал: Т стали статора 1 фаза (0..150 С)
	AI_03_RR(AI_K:= AI_K[0], AI_elpk04:=kontroller.AIn_[0]);
	// сигнал: Т стали статора 2 фаза (0..150 С)
	AI_03_RR(AI_K:= AI_K[1], AI_elpk04:=kontroller.AIn_[1]);
	// сигнал: Т стали статора 3 фаза (0..150 С)
	AI_03_RR(AI_K:= AI_K[2], AI_elpk04:=kontroller.AIn_[2]);
	// сигнал: Т меди статора 1 фаза (0..150 С)
	AI_03_RR(AI_K:= AI_K[3], AI_elpk04:=kontroller.AIn_[3]);
	// сигнал: Т меди статора 2 фаза (0..150 С)
	AI_03_RR(AI_K:= AI_K[4], AI_elpk04:=kontroller.AIn_[4]);
	// сигнал: Т меди статора 3 фаза (0..150 С)
	AI_03_RR(AI_K:= AI_K[5], AI_elpk04:=kontroller.AIn_[5]);
	// сигнал: Т ОП ЭД т.1 (0..100 С)
	AI_03_RR(AI_K:= AI_K[6], AI_elpk04:=kontroller.AIn_[6]);
	// сигнал: Т ОП ЭД со стороны редуктора т.2 (0..100 С)
	AI_03_RR(AI_K:= AI_K[7], AI_elpk04:=kontroller.AIn_[7]);
	// сигнал: Т ОП колеса редуктора со стороны ЭД т.3 (0..100 С)
	AI_03_RR(AI_K:= AI_K[8], AI_elpk04:=kontroller.AIn_[8]);
	// сигнал: Т ОП колеса редуктора со стороны Н т.4 (0..100 С)
	AI_03_RR(AI_K:= AI_K[9], AI_elpk04:=kontroller.AIn_[9]);
	// сигнал: Т ОП шестерни редуктора со стороны ЭД т.5 (0..100 С)
	AI_03_RR(AI_K:= AI_K[10], AI_elpk04:=kontroller.AIn_[10]);
	// сигнал: Т ОП шестерни редуктора со стороны Н т.6 (0..100 С)
	AI_03_RR(AI_K:= AI_K[11], AI_elpk04:=kontroller.AIn_[11]);
	// сигнал: Т ОП Н со стороны редуктора т.7, основной (0..100 С)
	AI_03_RR(AI_K:= AI_K[12], AI_elpk04:=kontroller.AIn_[12]);
	// сигнал: Т ОП Н со стороны редуктора т.7, резервный (0..100 С)
	AI_03_RR(AI_K:= AI_K[13], AI_elpk04:=kontroller.AIn_[13]);
	// сигнал: Т ОП Н со стороны своб.вала т.8, основной (0..100 С)
	AI_03_RR(AI_K:= AI_K[14], AI_elpk04:=kontroller.AIn_[14]);
	// сигнал: Т ОП Н со стороны своб.вала т.8, резервный (0..100 С)
	AI_03_RR(AI_K:= AI_K[15], AI_elpk04:=kontroller.AIn_[15]);

	
//////////////////////АНАЛОГОВЫЕ/////////////ПОЗ 13//////////////МАЦП-16//////////////////////////////////////////////////////

	// сигнал: Т ОП раб.колодок Н, т.9, основной (0..100 С)
	AI_03_RR(AI_K:= AI_K[16], AI_elpk04:=kontroller.AIn_[16]);
	// сигнал: Т ОП раб.колодок Н, т.9, резервный (0..100 С)
	AI_03_RR(AI_K:= AI_K[17], AI_elpk04:=kontroller.AIn_[17]);
	// сигнал: Т ОУП Н нераб.колодок, т.10, основной (0..100 С)
	AI_03_RR(AI_K:= AI_K[18], AI_elpk04:=kontroller.AIn_[18]);
	// сигнал: Т ОУП Н нераб.колодок, т.10, резервный (0..100 С)
	AI_03_RR(AI_K:= AI_K[19], AI_elpk04:=kontroller.AIn_[19]);
	// сигнал: Т холод.возд. в ЭД, т.1 (0..100 С)
	AI_03_RR(AI_K:= AI_K[20], AI_elpk04:=kontroller.AIn_[20]);
	// сигнал: Т холод.возд. в ЭД, т.2 (0..100 С)
	AI_03_RR(AI_K:= AI_K[21], AI_elpk04:=kontroller.AIn_[21]);
	// сигнал: Т горяч.возд. в ЭД, т.1 (0..100 С)
	AI_03_RR(AI_K:= AI_K[22], AI_elpk04:=kontroller.AIn_[22]);
	// сигнал: Т горяч.возд. в ЭД, т.2 (0..100 С)
	AI_03_RR(AI_K:= AI_K[23], AI_elpk04:=kontroller.AIn_[23]);
	// сигнал: Т наруж.возд. (РЕЗЕРВ)
	AI_03_RR(AI_K:= AI_K[24], AI_elpk04:=kontroller.AIn_[24]);
	// сигнал: Т газа на входе Н (-50..+100 С)
	AI_03_RR(AI_K:= AI_K[25], AI_elpk04:=kontroller.AIn_[25]);
	// сигнал: Т газа на выходе Н (-50..+100 С)
	AI_03_RR(AI_K:= AI_K[26], AI_elpk04:=kontroller.AIn_[26]);
	// сигнал: Т масла до АВОМ (0..+150 С)
	AI_03_RR(AI_K:= AI_K[27], AI_elpk04:=kontroller.AIn_[27]);
	// сигнал: Т масла после АВОМ (0..+150 С)
	AI_03_RR(AI_K:= AI_K[28], AI_elpk04:=kontroller.AIn_[28]);
	// сигнал: Т масла в МБ (0..+150 С)
	AI_03_RR(AI_K:= AI_K[29], AI_elpk04:=kontroller.AIn_[29]);
	// сигнал: Т масла в МБ над ТЭН (0..+100 С)
	AI_03_RR(AI_K:= AI_K[30], AI_elpk04:=kontroller.AIn_[30]);
	// сигнал: РЕЗЕРВ
	AI_03_RR(AI_K:= AI_K[31], AI_elpk04:=kontroller.AIn_[31]);

	
//////////////////////АНАЛОГОВЫЕ/////////////ПОЗ 11//////////////МАЦП-8//////////////////////////////////////////////////////

	// сигнал: Т в шкафу САУ (0..50 С)
	AI_03_RR(AI_K:= AI_K[32], AI_elpk04:=kontroller.AIn_[32]);
	// сигнал: P масла смазки низкое (0..0,4 МПа)
	AI_03_RR(AI_K:= AI_K[33], AI_elpk04:=kontroller.AIn_[33]);
	// сигнал: dP масла на масляном фильтре (0..250 кПа)
	AI_03_RR(AI_K:= AI_K[34], AI_elpk04:=kontroller.AIn_[34]);
	// сигнал: P масла смазки высокое (0..1 МПа)
	AI_03_RR(AI_K:= AI_K[35], AI_elpk04:=kontroller.AIn_[35]);
	// сигнал: P масла смазки после ГНС (0..1 МПа)
	AI_03_RR(AI_K:= AI_K[36], AI_elpk04:=kontroller.AIn_[36]);
	// сигнал: P масла после НУ (0..10 МПа)
	AI_03_RR(AI_K:= AI_K[37], AI_elpk04:=kontroller.AIn_[37]);
	// сигнал: РЕЗЕРВ
	AI_03_RR(AI_K:= AI_K[38], AI_elpk04:=kontroller.AIn_[38]);
	// сигнал: РЕЗЕРВ	
	AI_03_RR(AI_K:= AI_K[39], AI_elpk04:=kontroller.AIn_[39]);

	
//////////////////////АНАЛОГОВЫЕ/////////////ПОЗ 9//////////////МАЦП-8//////////////////////////////////////////////////////

	// сигнал: dP газа на конфузоре (0..0,25 МПа)
	AI_03_RR(AI_K:= AI_K[40], AI_elpk04:=kontroller.AIn_[40]);
	// сигнал: dP масло-газ (0..1,6 МПа)
	AI_03_RR(AI_K:= AI_K[41], AI_elpk04:=kontroller.AIn_[41]);
	// сигнал: Осевой сдвиг Н + (0..1 МПа)
	AI_03_RR(AI_K:= AI_K[42], AI_elpk04:=kontroller.AIn_[42]);
	// сигнал: Осевой сдвиг Н - (0..1 МПа)
	AI_03_RR(AI_K:= AI_K[43], AI_elpk04:=kontroller.AIn_[43]);
	// сигнал: Р газа на входе Н (0..10 МПа)
	AI_03_RR(AI_K:= AI_K[44], AI_elpk04:=kontroller.AIn_[44]);
	// сигнал: Р газа на выходе Н (0..10 МПа)
	AI_03_RR(AI_K:= AI_K[45], AI_elpk04:=kontroller.AIn_[45]);
	// сигнал: Р имп.газа (0..10 МПа)
	AI_03_RR(AI_K:= AI_K[46], AI_elpk04:=kontroller.AIn_[46]);
	// сигнал: РЕЗЕРВ
	AI_03_RR(AI_K:= AI_K[47], AI_elpk04:=kontroller.AIn_[47]);

	
//////////////////////АНАЛОГОВЫЕ/////////////ПОЗ 16//////////////МАЦП-8//////////////////////////////////////////////////////

	// сигнал: Уровень масла в маслобаке (200..885 мм)
	AI_03_RR(AI_K:= AI_K[48], AI_elpk04:=kontroller.AIn_[48]);
	// сигнал: РЕЗЕРВ
	AI_03_RR(AI_K:= AI_K[49], AI_elpk04:=kontroller.AIn_[49]);
	// сигнал: РЕЗЕРВ
	AI_03_RR(AI_K:= AI_K[50], AI_elpk04:=kontroller.AIn_[50]);
	// сигнал: РЕЗЕРВ
	AI_03_RR(AI_K:= AI_K[51], AI_elpk04:=kontroller.AIn_[51]);
	// сигнал: Контроль ~220 САУ (0..250 В)
	AI_03_RR(AI_K:= AI_K[52], AI_elpk04:=kontroller.AIn_[52]);
	// сигнал: Контроль =220 САУ (0..250 В)
	AI_03_RR(AI_K:= AI_K[53], AI_elpk04:=kontroller.AIn_[53]);
	// сигнал: РЕЗЕРВ
	AI_03_RR(AI_K:= AI_K[54], AI_elpk04:=kontroller.AIn_[54]);
	// сигнал: РЕЗЕРВ
	AI_03_RR(AI_K:= AI_K[55], AI_elpk04:=kontroller.AIn_[55]);
	
	
//////////////////////АНАЛОГОВЫЕ/////////////ПОЗ 14//////////////МАЦП-8//////////////////////////////////////////////////////

	// сигнал: Виброскорость ОП ЭД, т.1 (0..25 мм/сек)
	AI_03_RR(AI_K:= AI_K[56], AI_elpk04:=kontroller.AIn_[56]);
	// сигнал: Виброскорость ОУП ЭД со стороны редуктора, т.2 (0..25 мм/сек)
	AI_03_RR(AI_K:= AI_K[57], AI_elpk04:=kontroller.AIn_[57]);
	// сигнал: Виброскорость ОУП колеса редуктора со стороны ЭД, т.3 (0..25 мм/сек)
	AI_03_RR(AI_K:= AI_K[58], AI_elpk04:=kontroller.AIn_[58]);
	// сигнал: Виброскорость ОП колеса редуктора со стороны Н, т.4 (0..25 мм/сек)
	AI_03_RR(AI_K:= AI_K[59], AI_elpk04:=kontroller.AIn_[59]);
	// сигнал: Виброскорость ОП шестерни редуктора со стороны ЭД, т.5 (0..25 мм/сек)
	AI_03_RR(AI_K:= AI_K[60], AI_elpk04:=kontroller.AIn_[60]);
	// сигнал: Виброскорость ОП шестерни редуктора со стороны Н, т.6 (0..25 мм/сек)
	AI_03_RR(AI_K:= AI_K[61], AI_elpk04:=kontroller.AIn_[61]);
	// сигнал: Виброперемещение вала Н со стороны редуктора, т.7 (0..125 мкм)
	AI_03_RR(AI_K:= AI_K[62], AI_elpk04:=kontroller.AIn_[62]);
	// сигнал: Виброперемещение вала Н, т.8 (0..125 мкм)   РЕЗЕРВ
	AI_03_RR(AI_K:= AI_K[63], AI_elpk04:=kontroller.AIn_[63]);
	
	
//////////////////////АНАЛОГОВЫЕ/////////////ПОЗ 12//////////////МАЦП-8//////////////////////////////////////////////////////

	// сигнал: РЕЗЕРВ
	AI_03_RR(AI_K:= AI_K[64], AI_elpk04:=kontroller.AIn_[64]);
	// сигнал: Ток статора (помпаж), (0..1000 А)
	AI_03_RR(AI_K:= AI_K[65], AI_elpk04:=kontroller.AIn_[65]);
	// сигнал: РЕЗЕРВ
	AI_03_RR(AI_K:= AI_K[66], AI_elpk04:=kontroller.AIn_[66]);
	// сигнал: РЕЗЕРВ
	AI_03_RR(AI_K:= AI_K[67], AI_elpk04:=kontroller.AIn_[67]);
	// сигнал: РЕЗЕРВ
	AI_03_RR(AI_K:= AI_K[68], AI_elpk04:=kontroller.AIn_[68]);
	// сигнал: РЕЗЕРВ
	AI_03_RR(AI_K:= AI_K[69], AI_elpk04:=kontroller.AIn_[69]);
	// сигнал: РЕЗЕРВ
	AI_03_RR(AI_K:= AI_K[70], AI_elpk04:=kontroller.AIn_[70]);
	// сигнал: РЕЗЕРВ
	AI_03_RR(AI_K:= AI_K[71], AI_elpk04:=kontroller.AIn_[71]);

END_PROGRAM

// Elpk_03_02_COMMON/DI_03_R
FUNCTION DI_03_R : WORD
VAR_INPUT
	DI_K0:	BOOL{T_DI03};	
	DIb_K0:	BOOL{T_DI03};
	N_Pair: WORD;	// 1..8	
END_VAR
VAR_IN_OUT
	K_OUT:WORD;
END_VAR
VAR_OUTPUT
//	DI_OUT:	BOOL{T_DI03};	
//	DIb_OUT:BOOL{T_DI03};	
END_VAR


VAR
END_VAR


//	kontroller.DIn_[0].val.0	:=		DI_K[0].In.0:=1;	// сигнал: Кран 1 открыт
//	kontroller.DIn_[0].val.1	:=		1;				// обрыв: Нет обрыва

//	kontroller.DIn_[4].val.0	:=		DI_K[2].In.0:=1;	// сигнал: dP масло-газ < 100 кПА
//	kontroller.DIn_[4].val.1	:=		DI_K[2].In.1:=1;	// обрыв:  dP масло-газ < 100 кПА

	//DI_OUT:=	DI_K0;		// сигнал: аналоговый сигнал	
	//DIb_OUT:=	DIb_K0;		// обрыв: Есть обрыв или Нет обрыва	

	CASE N_Pair OF
	1:
		K_OUT.0:=	DI_K0;		// сигнал: аналоговый сигнал
		K_OUT.1:=	DIb_K0;		// обрыв: Есть обрыв или Нет обрыва
	2:
		K_OUT.2:=	DI_K0;		// сигнал: аналоговый сигнал
		K_OUT.3:=	DIb_K0;		// обрыв: Есть обрыв или Нет обрыва
	3:
		K_OUT.4:=	DI_K0;		// сигнал: аналоговый сигнал
		K_OUT.5:=	DIb_K0;		// обрыв: Есть обрыв или Нет обрыва
	4:
		K_OUT.6:=	DI_K0;		// сигнал: аналоговый сигнал
		K_OUT.7:=	DIb_K0;		// обрыв: Есть обрыв или Нет обрыва
	5:
		K_OUT.8:=	DI_K0;		// сигнал: аналоговый сигнал
		K_OUT.9:=	DIb_K0;		// обрыв: Есть обрыв или Нет обрыва
	6:
		K_OUT.10:=	DI_K0;		// сигнал: аналоговый сигнал
		K_OUT.11:=	DIb_K0;		// обрыв: Есть обрыв или Нет обрыва
	7:
		K_OUT.12:=	DI_K0;		// сигнал: аналоговый сигнал
		K_OUT.13:=	DIb_K0;		// обрыв: Есть обрыв или Нет обрыва
	8:
		K_OUT.14:=	DI_K0;		// сигнал: аналоговый сигнал
		K_OUT.15:=	DIb_K0;		// обрыв: Есть обрыв или Нет обрыва

	END_CASE

END_FUNCTION

// Elpk_03_02_COMMON/AI_03_RR
FUNCTION AI_03_RR : WORD
VAR_IN_OUT
	AI_K:	T_AI03;	
//	K	:	elpk04;
	AI_elpk04	:	AIn_s;
END_VAR
VAR
END_VAR


	AI_elpk04.f	:=	5;					// .0 - есть в проекте		.1 - входные		.2 - достоверность	

	IF (AI_K.Imx=16#55AA) THEN
		AI_K.RR:=AI_K.Im;
		//AI_elpk04.f.2	:=	AI_K.VeraB;		// достоверность из драйвера RWH (=1 - достоверно)	
	ELSE
		AI_K.RR:=AI_K.In;
		AI_elpk04.f.2	:=	AI_K.VeraB;		// достоверность из драйвера RWH (=1 - достоверно)	
	END_IF
		AI_elpk04.val	:=	AI_K.RR;		// сигнал: аналоговый сигнал

END_FUNCTION

// lowLevel_ecl/kontroller/mlp/Elpk04
{attribute 'symbol' := 'none'}
FUNCTION_BLOCK Elpk04 EXTENDS baseKontroller
VAR_INPUT
	mlpConfig:STRING;

	DIn_ 	:	ARRAY [0..255] 	OF DIn_s;		//	Сигнализация и неисправности дискретных входов (номер в массиве соответствует адресу конфигурации в MLP)
											//	f	:	WORD	;	//	bit-0 присутствие в проекте MLP. 1-есть, 0 -нет
																	//	bit-1 тип модуля 1-выходной, 0 -входной
																	//	bit-2 достоверность 1- достоверно,0- не достоверно 
											//	val	:	WORD	;	//	Контроль канала
																	//	Каждая цепь 2 бита
	                												//	00 - обыв цепи
																	//	01 - недостоверно
																	//	10 - контакт разомкнут
																	//	11 - контакт замкнут	

											//	DIn[63].val - меняющееся число для проверки связи с основным МЛП (задается в MLP)
											//	если	DIn[64].val = 7 - есть связь с BS-1 (задается в MLP)
											//	если	DIn[65].val = 7 - есть связь с BS-2 (задается в MLP)
											//	если	DIn[66].val = 7 - есть связь с BS-3 (задается в MLP)
											//	если	DIn[67].val = 7 - есть связь с BS-4 (задается в MLP)
																					
																	
AIn_ 	:	ARRAY [0..255] 	OF AIn_s;		//	Значение и неисправности аналоговых входов (номер в массиве соответствует адресу конфигурации в MLP)
											//	f	:	DWORD	;	//	bit-0 присутствие в проекте MLP. 1-есть, 0 –нет
																	//	bit-1 тип модуля 1-выходной, 0 -входной
																	//	bit-2 достоверность 1- достоверно,0- не достоверно. Диагностика общая: и по диапазонам измерения, и собственная по каналу модуля.
																	//	bit-3 размерность сигнала 1- в физических величинах,0- значение тока (0-20100)
																	//	bit-4 1- ниже нижней границы,0 - выше нижней границы
																	//	bit-5 1- выше верхней границы,0 - ниже верхней границы
																	//	bit-6 1- общий бит отказа канала( по ИЛИ Not(bit2), bit4, bit5)
											//	val	:	REAL	;	//	Значение аналогового входа 4-20мА - 40000-20000 

Dout_	:	ARRAY [0..255] 	OF WORD;		//	Массив дискретных выходов (один бит - один выход, одно слово - один модуль) (номер в массиве соответствует адресу конфигурации в MLP)
Din_Dout: 	ARRAY [0..255] 	OF sDIN_DOUT;	//	Массив неисправностей дискретных выходов
											//	s_Aux	:	WORD	;	//	bit-0 присутствие 1-есть, 0 -нет (привязка в конфигурации MLP)
																		//	bit-1 тип модуля 1-выходной, 0 -входной
																		//	bit-2 достоверность 1- достоверно,0- не достоверно
									  		//	kcc		:	WORD	;   //	Контроль Целостности Цепи - КЦЦ
																		//	каждая цепь 2 бита
																		//	00 - неизвестно или обрыв цепи
																		//	01 - есть Целостность Цепи
																		//	10 - есть ток
																		//	11 - КЗ
											//	kk		:	WORD	;	//	Контроль выхода команды - КК
																		//	каждая цепь 2 бита
																		//	00 - не бывает
																		//	01 - пассивное состояние
																		//	10 - активное (есть выход)состояние
																		//	11 - ошибка выхода команды 
									  		//	value_cc:	WORD	;	//	содержимое выходных регистров 

Aout_ 	:	ARRAY [0..255] 	OF REAL;		//	Массив аналоговых выходов (номер в массиве соответствует адресу конфигурации в MLP)
Ain_Aout:	ARRAY [0..255] 	OF sAIN_AOUT;	//	Массив неисправностей аналоговых выходов
											//	s_Aux	:	WORD	;	//	bit-0 присутствие 1-есть, 0 -нет
																		//	bit-1 тип модуля 1-выходной, 0 -входной
																		//	bit-2 достоверность 1- достоверно,0- не достоверно
																		//	s_value	:	REAL	;	//	Действительный (измеренный) выходной ток 4-20мА - 4000-20000

Diag_ 	:	ARRAY [0..63]	OF WORD;		//	массив неисправностей модулей
																		//	2 бита на 1 модуль
																		//	00 - ok
																		//	01 - нет модуля
																		//	10 - нулевые данные
		

														//	11 - нет связи с модулем
END_VAR
VAR_OUTPUT
	{attribute 'symbol' := 'read'}
	Diagnostic:DiagnosticMlp:=(elpk:=THIS);
END_VAR
VAR
	_init:BOOL;
END_VAR

SUPER^();
IF NOT _init THEN
///	Diagnostic.readConfig(mlpConfig:=mlpConfig);
	Diagnostic.readConfig_faleev(mlpConfig:=mlpConfig);
	callSetController(table:=inputTable);
	callSetController(table:=outputTable);
	_init:=TRUE;
END_IF

Diagnostic();

METHOD PRIVATE callSetController
VAR_INPUT
	CONSTANT table:TableDescriptor;
END_VAR
VAR
	curObject:POINTER TO BaseObject;
	curSource:IMlpSource;
END_VAR
curObject:=table.head;
IF curObject=0 THEN
	RETURN;
END_IF
REPEAT
	IF (__QUERYINTERFACE(curObject^,curSource)) THEN		
		curSource.setKontroller(THIS^);
	END_IF;
	curObject:=curObject^.getNext();
	UNTIL curObject=0
END_REPEAT
END_METHOD

END_FUNCTION_BLOCK

// lowLevel_ecl/kontroller/baseKontroller
	{attribute 'symbol' := 'none'}
FUNCTION_BLOCK baseKontroller EXTENDS BaseObject
IMPLEMENTS IKontroller
VAR_INPUT
END_VAR
VAR_OUTPUT
END_VAR
VAR_IN_OUT
END_VAR
VAR
	{attribute 'symbol' := 'none'}
	inputTable:TableDescriptor;
	{attribute 'symbol' := 'none'}
	outputTable:TableDescriptor;	
	{attribute 'symbol' := 'readwrite'}
	imit:BOOL;
	
	_imitTrig: RP_trig;
END_VAR

SUPER^();

_imitTrig(in:=imit);
IF _imitTrig.Qp OR _imitTrig.Qn THEN
	setImit(table:=inputTable,nimit:=imit);
	setImit(table:=outputTable,nimit:=imit);
END_IF

METHOD callOutputTable
VAR_INPUT
END_VAR
callExec(OutputTable);
END_METHOD

METHOD PRIVATE setImit
VAR_INPUT
	table:TableDescriptor;
	nimit:BOOL;
END_VAR
VAR
	curObject:POINTER TO BaseObject;
	curSource:ISource;
END_VAR
curObject:=table.head;
IF curObject=0 THEN
	RETURN;
END_IF
REPEAT
	IF (__QUERYINTERFACE(curObject^,curSource)) THEN		
			curSource.imit:=nimit;
	END_IF;
	curObject:=curObject^.getNext();
	UNTIL curObject=0
END_REPEAT
END_METHOD

METHOD PUBLIC callCommands
VAR_INPUT
END_VAR
ExecComands(table:=inputTable);
ExecComands(table:=outputTable);
END_METHOD

METHOD PUBLIC callInputTable
VAR_INPUT
END_VAR
callExec(inputTable);
END_METHOD

END_FUNCTION_BLOCK

// lowLevel_ecl/Common/BaseObject
	{attribute 'symbol' := 'none'}
	{attribute 'reflection'}
FUNCTION_BLOCK BaseObject
IMPLEMENTS __SYSTEM.IQueryInterface
VAR_INPUT		

END_VAR
VAR_OUTPUT
END_VAR
VAR
	_next:POINTER TO BaseObject;
	
	fileHandle:RTS_IEC_HANDLE;
	initialized:BOOL;
	PersistWrited:BOOL;	
	hawePersist:BOOL;
	
	{attribute 'instance-path'} 
	{attribute 'noinit'} 
	name: STRING; 
END_VAR
VAR_STAT
	ForseWritePersist:BOOL;//=true-Сохраняет Persistent переменные всех объектов в проекте
END_VAR

IF NOT initialized THEN	
	LoadFromFile();
	initialized:=TRUE;
	registerInAcrhive();
	onInit();
END_IF

IF ForseWritePersist THEN
	IF NOT PersistWrited THEN
		SaveToFile();
		PersistWrited:=TRUE;
	END_IF
ELSE
	PersistWrited:=FALSE;
END_IF

METHOD FB_init : BOOL
VAR_INPUT
  bInitRetains : BOOL; // if TRUE, the retain variables are initialized (warm start / cold start)
  bInCopyCode : BOOL;  // if TRUE, the instance afterwards gets moved into the copy code (online change)
  table: POINTER TO TableDescriptor;
END_VAR
IF (table<>0) THEN
	IF (table^.head=0)THEN
		table^.head:=THIS;
		table^.tail:=THIS;
		_next:=0;
	ELSE
		table^.tail^._next:=THIS;
		_next:=0;
		table^.tail:=THIS;
	END_IF
END_IF;
END_METHOD

METHOD getNext : POINTER TO BaseObject
VAR_INPUT
END_VAR
getNext:=_next;
END_METHOD

METHOD PROTECTED setDefaultPersistent:BOOL
VAR_INPUT
END_VAR
setDefaultPersistent:=FALSE;
END_METHOD

METHOD FINAL SaveToFile
VAR_INPUT
END_VAR
VAR
	fileName:STRING(255);
	res1:DWORD;
	pres1:POINTER TO rts_iec_result:=ADR(res1);
END_VAR
VAR CONSTANT
	dirName:STRING:='\storage card\3s\persist\';
END_VAR
fileName:=CONCAT(dirname,CONCAT(name,'.pss'));
fileHandle:=SysFileopen(szfile:=filename, am:=am_write, presult:=pres1);
IF (fileHandle<>0)AND(res1=0) THEN
	hawePersist:=FALSE;
	writePersistent();
	//SysFileStreamFClose(File:=fileHandle);
	sysfileClose(filehandle);
	fileHandle:=0;
	IF NOT hawePersist THEN
		//SysFileStreamRemove(FileName);
		sysfiledeletebyhandle(hfile:=filehandle);
	END_IF
END_IF
END_METHOD

METHOD PRIVATE LoadFromFile
VAR_INPUT
END_VAR
VAR
	fileName:STRING(255);
	res1:DWORD;
	pres1:POINTER TO rts_iec_result:=ADR(res1);
END_VAR
VAR CONSTANT
	dirname:STRING:='\storage card\3s\persist\';
END_VAR
fileName:=CONCAT(dirname,CONCAT(name,'.pss'));
fileHandle:=SysFileStreamFopen(FileName:=filename,mode:='r');
IF (fileHandle<>0) THEN
	readPersistent();
	sysfileStreamFClose(File:=filehandle);
	fileHandle:=0;
ELSE
	IF setDefaultPersistent() THEN
		SaveToFile();
	END_IF
END_IF
END_METHOD

METHOD PROTECTED readPersistent
VAR_INPUT
END_VAR
END_METHOD

METHOD PROTECTED writePersistent
VAR_INPUT
END_VAR
END_METHOD

METHOD PROTECTED writeValue
VAR_INPUT
	value:STRING;
	comment:STRING;
END_VAR
VAR CONSTANT
	komment:STRING:='//';
	endln:STRING:='$N';
END_VAR
VAR
	s1:STRING(255);
	res1:DWORD;
	pres1:POINTER TO rts_iec_result:=ADR(res1);
	
END_VAR
s1:=concat(value, komment);
s1:=concat(s1,comment);
s1:=concat(s1,endln);
sysfilewrite(hfile:=filehandle,pbybuffer:=ADR(s1),ulsize:=len(s1),presult:=pres1);



hawePersist:=TRUE;
(*SysFileStreamFPutS (File:=fileHandle,str:=ADR(value));
SysFileStreamFPutS (File:=fileHandle,str:=ADR(komment));
SysFileStreamFPutS (File:=fileHandle,str:=ADR(comment));
SysFileStreamFPutS (File:=fileHandle,str:=ADR(endln));*)
END_METHOD

METHOD PROTECTED readValue : String
VAR_INPUT
END_VAR
VAR
	cStr:STRING;
	strPos:INT;
	res1:DWORD;
	pres1:pointer to rts_iec_result:=adr(res1);
END_VAR
sysfileStreamFGetS(str:=ADR(cStr),n:=SIZEOF(cStr), File:=fileHandle);
strPos:=FIND(STR1:=cStr,STR2:='//');
IF strPos =0 THEN
	strPos:=FIND(STR1:=cStr,STR2:='$N');
END_IF
IF strPos<>0 THEN
	readValue:=LEFT(STR:=cStr,SIZE:=strPos-1);
ELSE
	readValue:=cStr;		
END_IF
END_METHOD

METHOD PROTECTED onInit
VAR_INPUT
END_VAR
END_METHOD

METHOD PRIVATE registerInAcrhive
VAR_INPUT
END_VAR
VAR
	provider:ArchiveProvider;
END_VAR
provider.RegisterSource(object:= THIS);
END_METHOD

END_FUNCTION_BLOCK

// lowLevel_ecl/EmergencyAarchive/ArchiveProvider
FUNCTION_BLOCK ArchiveProvider
VAR_INPUT
END_VAR
VAR_OUTPUT
END_VAR
VAR
END_VAR
VAR_STAT
	archiveInst: POINTER TO Archive;
END_VAR

METHOD PUBLIC RegisterArchive
VAR_INPUT
	nArchive:pointer TO Archive;
END_VAR
archiveInst := nArchive;
END_METHOD

METHOD RegisterSource
VAR_INPUT
	object: POINTER TO BaseObject;
END_VAR
IF (archiveInst<>0) THEN
	archiveInst^.appendSource(object);
END_IF
END_METHOD

METHOD PUBLIC accidentStarted
VAR_INPUT
	descript:STRING;
END_VAR
IF (archiveInst<>0) THEN
	archiveInst^.startAccident(descript);
END_IF
END_METHOD

END_FUNCTION_BLOCK

// lowLevel_ecl/EmergencyAarchive/Archive
	{attribute 'symbol' := 'none'}
FUNCTION_BLOCK Archive EXTENDS BaseObject
VAR_INPUT
	recordDuration:TIME:=T#5M;	
	writeFileTimeKvant:TIME:=T#250MS;
	dirName:STRING:= '.\archive\';
END_VAR
VAR_OUTPUT
END_VAR
VAR
	TimeSlices:LAT.List;
	provider:ArchiveProvider;
	
	accidentStarted:BOOL;
	accidentStartedTrig:R_TRIG;
	currentLogName:STRING;
	accidentTime:SYSTIME;
	lastSavedTimeStamp:SYSTIME;
	accidentDesc:STRING;
	memoryError:BOOL;
	
	archiveFileHandle:RTS_IEC_HANDLE;
	currentWritedSlice:LAT.IElement;
END_VAR
VAR_TEMP
	newTimeSlice:POINTER TO TimeSlice;
	newTimeSliceInterface: LAT.IElement;
	
	now:SYSTIME;
	lastTime:SYSTIME;
	lastSliceTime:SYSTIME;
	
END_VAR
VAR CONSTANT
	devisor:STRING:=';';
	endln:STRING:='$n';
END_VAR

IF (TimeSlices.ListIsEmpty) THEN
	RETURN;
END_IF

SysTimeRtcHighResGet(pTimestamp:= now);
lastTime:= now-TIME_TO_ULINT(recordDuration);
lastSliceTime:=firstTimeSlice^.timeStamp;

IF (lastSliceTime<lastTime) OR memoryError THEN
	newTimeSlice:=firstTimeSlice;
	newTimeSliceInterface:=TimeSlices.PopElem();
	TimeSlices.AppendElem(newTimeSliceInterface);
	newTimeSlice^.update();
ELSE	
	newTimeSlice:=lastTimeSlice^.copy();
	IF (newTimeSlice <>0) THEN
		IF __QUERYINTERFACE(newTimeSlice^,newTimeSliceInterface) THEN
			TimeSlices.AppendElem(newTimeSliceInterface);
			newTimeSlice^.update();
		ELSE
			__DELETE(newTimeSlice);
		END_IF
	ELSE
		memoryError:=TRUE;
	END_IF
END_IF

IF archiveFileHandle<>0 THEN
	countinueDataWrite();
END_IF
accidentStartedTrig(CLK:=accidentStarted);
IF accidentStartedTrig.Q THEN
	currentLogName:=CONCAT(dirName,concat(timeToFileName(accidentTime),'.csv'));
	lastSavedTimeStamp:=lastTimeSlice^.timeStamp;
	writeLog(currentLogName,FALSE);
ELSE	
	IF accidentStarted THEN 
		IF (firstTimeSlice^.timeStamp>lastSavedTimeStamp) THEN
		lastSavedTimeStamp:=lastTimeSlice^.timeStamp;
		writeLog(currentLogName,TRUE);
		accidentStarted:=FALSE;
		END_IF
	END_IF
END_IF

METHOD PUBLIC appendSource
VAR_INPUT
	object: POINTER TO BaseObject;
END_VAR
VAR
	currentSlice:LAT.IElement;
	pCurrentSlice: POINTER TO TimeSlice;
	newListener:IObjectListener;
END_VAR
IF TimeSlices.ListIsEmpty THEN
	newTimeSlice();
END_IF

IF NOT TimeSlices.ListIsEmpty THEN
	currentSlice:=TimeSlices.HeadElem;		
	REPEAT
		__QUERYPOINTER (currentSlice,pCurrentSlice);
		IF  createObjectListener(object:=object,newListener=>newListener) THEN
			IF newListener<>0 THEN
				pCurrentSlice^.appendValueListener(newListener);
			ELSE
				LogAdd(CmpLog.STD_LOGGER,'EmergencyAarchive',UDINT_TO_DINT(CmpLog.LogClass.LOG_ERROR),0,0,'Not enough dynamic memory for new object.');
			END_IF			
		ELSE
			RETURN;
		END_IF
		currentSlice:=currentSlice.NextElem;
	UNTIL 	currentSlice =0
	END_REPEAT	
END_IF
END_METHOD

METHOD PRIVATE newTimeSlice
VAR_INPUT
END_VAR
VAR
	newTimeSlice: POINTER TO TimeSlice;
	newTimeSliceInterface: LAT.IElement;
	timeStamp:SYSTIME:=0;
END_VAR
newTimeSlice:=__NEW(TimeSlice);
IF (newTimeSlice<>0) THEN
	SysTimeRtcHighResGet(pTimestamp:=timeStamp);
	newTimeSlice^.timeStamp:=timeStamp;
	IF __QUERYINTERFACE(newTimeSlice^,newTimeSliceInterface) THEN
		TimeSlices.AppendElem(newTimeSliceInterface);
	ELSE
		__DELETE(newTimeSlice);
	END_IF
END_IF
END_METHOD

PROPERTY PRIVATE lastTimeSlice : pointer to TimeSlice
GET
lastTimeSlice:=0;
IF TimeSlices.ListIsEmpty THEN
	RETURN;
END_IF

__QUERYPOINTER(TimeSlices.TailElem,lastTimeSlice);
END_GET
END_PROPERTY

PROPERTY PRIVATE firstTimeSlice : pointer to TimeSlice
GET
firstTimeSlice:=0;
IF TimeSlices.ListIsEmpty THEN
	RETURN;
END_IF

__QUERYPOINTER(TimeSlices.HeadElem,firstTimeSlice);
END_GET
END_PROPERTY

METHOD PRIVATE timeToString : String
VAR_INPUT
	hrTime:SYSTIME;
END_VAR
VAR
	 unpTime:SYSTIMEDATE;
END_VAR
///SysTimeRtcConvertHighResToLocal(pTimestamp:=hrTime,pDate:=unpTime);

 timeToString:=CONCAT(uintToStrf(unpTime.wYear,4),'-');
 timeToString:=CONCAT(timeToString,uintToStrf(unpTime.wMonth,2));
 timeToString:=CONCAT(timeToString,'-');
 timeToString:=CONCAT(timeToString,uintToStrf(unpTime.wDay,2));
 timeToString:=CONCAT(timeToString,'T');
 timeToString:=CONCAT(timeToString,uintToStrf(unpTime.wHour,2));
 timeToString:=CONCAT(timeToString,':');
 timeToString:=CONCAT(timeToString,uintToStrf(unpTime.wMinute,2));
 timeToString:=CONCAT(timeToString,':');
 timeToString:=CONCAT(timeToString,uintToStrf(unpTime.wSecond,2));
 timeToString:=CONCAT(timeToString,',');
 timeToString:=CONCAT(timeToString,uintToStrf(unpTime.wMilliseconds,3));
END_METHOD

METHOD PRIVATE timeTofileName : String
VAR_INPUT
	hrTime:SYSTIME;
END_VAR
VAR
	 unpTime:SYSTIMEDATE;
END_VAR
 ///SysTimeRtcConvertHighResToLocal(pTimestamp:=hrTime,pDate:=unpTime);

 timeTofileName:=CONCAT(uintToStrf(unpTime.wYear,4),'-');
 timeTofileName:=CONCAT(timeTofileName,uintToStrf(unpTime.wMonth,2));
 timeTofileName:=CONCAT(timeTofileName,'-');
 timeTofileName:=CONCAT(timeTofileName,uintToStrf(unpTime.wDay,2));
 timeTofileName:=CONCAT(timeTofileName,'_');
 timeTofileName:=CONCAT(timeTofileName,uintToStrf(unpTime.wHour,2));
 timeTofileName:=CONCAT(timeTofileName,'_');
 timeTofileName:=CONCAT(timeTofileName,uintToStrf(unpTime.wMinute,2));
 timeTofileName:=CONCAT(timeTofileName,'_');
 timeTofileName:=CONCAT(timeTofileName,uintToStrf(unpTime.wSecond,2));
END_METHOD

METHOD PRIVATE uintToStrf : STRING
VAR_INPUT
	val:UINT;
	size:INT;
END_VAR
VAR
	startLength:int;
	i:INT;
END_VAR
uintToStrf:=UINT_TO_STRING(val);
startLength:=LEN(uintToStrf);
IF startLength<size THEN
	FOR i:=startLength TO size-1 DO
		uintToStrf:=CONCAT('0',uintToStrf);
	END_FOR
END_IF
END_METHOD

METHOD PRIVATE writeHead
VAR_INPUT
	h_file:RTS_IEC_HANDLE;
END_VAR
VAR
	curData:STRING;
	currentObject: LAT.IElement;
	pCurrentObject:IObjectListener;	
	parameterIndex:WORD;
	parameterCount:WORD;	
END_VAR
curData:=timeToString(hrTime:=accidentTime);
SysFileStreamFPutS(File:=h_file,str:=ADR(curData));	
SysFileStreamFPutS(File:=h_file,str:=ADR(devisor));
SysFileStreamFPutS(File:=h_file,str:=ADR(accidentDesc));
SysFileStreamFPutS(File:=h_file,str:=ADR(endln));

IF NOT lastTimeSlice^.values.ListIsEmpty THEN
	currentObject:=lastTimeSlice^.values.HeadElem;
	REPEAT
		__QUERYINTERFACE (currentObject,pCurrentObject);
		curData:=pCurrentObject.getName();
		SysFileStreamFPutS(File:=h_file,str:=ADR(devisor));
		SysFileStreamFPutS(File:=h_file,str:=ADR(curData)); 
		
		parameterCount:= pCurrentObject.getParametersCount();
		IF parameterCount>1 THEN
			FOR parameterIndex:=2 TO parameterCount DO
				SysFileStreamFPutS(File:=h_file,str:=ADR(devisor));			
			END_FOR
		END_IF			
		currentObject:=currentObject.NextElem;
	UNTIL 	currentObject =0
	END_REPEAT
	
	SysFileStreamFPutS(File:=h_file,str:=ADR(endln));
	
	currentObject:=lastTimeSlice^.values.HeadElem;
	REPEAT
		__QUERYINTERFACE (currentObject,pCurrentObject);
		
